(* CoDeSys 2.3 library: TcMC2.lib *)
(* Libraries: STANDARD.LIB 5.6.98 11:03:02, TcBase.lib*14.5.09 11:14:08, TcSystem.lib*15.1.10 08:10:33, TcBaseMath.lib 27.7.04 11:07:56, TcMath.lib 23.9.04 14:15:30 *)

(* Global variable list: TcMC_GlobalConstants *)
VAR_GLOBAL
	TcMcGlobal : _TCMCGLOBAL;
END_VAR
VAR_GLOBAL CONSTANT
	DEFAULT_HOME_POSITION 	:	LREAL 	:= 1.0E307;
END_VAR

(* Data type *)
{library private}
TYPE _E_ParameterType :
 (
	PARAMETERTYPE_NOTYPE := 0,
	PARAMETERTYPE_BOOL,
	PARAMETERTYPE_DWORD,
	PARAMETERTYPE_LREAL
 );
END_TYPE

(* Data type *)
{library private}
TYPE _E_ReadWriteParameterMode :
 (
	READWRITEPARAMETERMODE_READ 	:=10,
	READWRITEPARAMETERMODE_WRITE	:= 11
 );
END_TYPE

(* Data type *)
{library private}
TYPE _E_TcMC_STATES :
 (
	STATE_INITIALIZATION  := 100,
	STATE_ORDER,
	STATE_RUNNING,
	STATE_WAITING,
	STATE_MOTIONCOMMANDSLOCKED
 );
END_TYPE

(* Data type *)
TYPE _E_TcNC_CmdState :
 (
	CMDSTATE_SUCCESSFULLY_EXECUTED				:= 1,	(* bit number *)
	CMDSTATE_ABORTED_WITHOUT_ERROR				:= 2,
	CMDSTATE_ENDED_WITH_ERROR					:= 3,
	CMDSTATE_LASTCMD_SUCCESSFULLY_EXECUTED	:= 8,
	CMDSTATE_LASTCMD_ABORTED_WITHOUT_ERROR	:= 9,
	CMDSTATE_LASTCMD_ENDED_WITH_ERROR			:= 10
 );
END_TYPE

(* Data type *)
TYPE _E_TcNC_CmdTypeNewTargPosAndVelo :
 (
	TCNC_CHANGE_POS						:=  1,		(*Position (instantan)*)
	TCNC_CHANGE_VELO,							(*Geschwindigkeit (instantan)*)
	TCNC_CHANGE_POSANDVELO,					(*Position und Geschwindigkeit (instantan)*)
	TCNC_CHANGE_POS_AT_SWITCHPOS		:=  9,		(*Position (Umschaltposition)*)
	TCNC_CHANGE_VELO_AT_SWITCHPOS,			(*Geschwindigkeit (Umschaltposition)*)
	TCNC_CHANGE_POSANDVELO_AT_SWITCHPOS,	(*Position und Geschwindigkeit (Umschaltposition)*)
	TCNC_REACH_VELO_AT_POS				:= 14		(*neue Geschwindigkeit wird an einer bestimmten Position erreicht *)
 );
END_TYPE

(* Data type *)
TYPE _E_TcNC_PosSetType : (* mode is used with MC_SetPosition *)
(
	TCNC_POSSETTYPE_ABSOLUTE		:= 1,	(*Absolute position*)
	TCNC_POSSETTYPE_RELATIVE			(*Relative position*)
);
END_TYPE

(* Data type *)
TYPE _E_TcNC_ServoState :
 (
	TCNC_INACTIVE 	:= 0,
	TCNC_RUNNING,
	TCNC_OVERRIDE_ZERO,
	TCNC_PHASE_VELOCONST,
	TCNC_PHASE_ACCPOS,
	TCNC_PHASE_ACCNEG
 );
END_TYPE

(* Data type *)
TYPE _E_TcNC_SlaveTypes :
(
	TCNC_SLAVETYPE_LINEAR							:=	1,	(* Lineare Kopplung (Geradengleichung) *)
	TCNC_SLAVETYPE_FLYINGSAW_ONVELOCITY		:= 	2,	(* diagonal synchron. Aufkoppeln schnellstens auf Geschwindigkeit *)
	TCNC_SLAVETYPE_FLYINGSAW_ONPOSITION		:=	3,	(* diagonal synchron. Aufkoppeln auf Position und Geschwindigkeit *)
	TCNC_SLAVETYPE_FLYINGSAW_QUADRATIC		:=	4,	(* diagonal synchron. Aufkoppeln (quadratisches Geschw.-Profil) *)
	TCNC_SLAVETYPE_SYNCHRONIZING_ONVELO		:= 	5,	(* synchron. Aufkoppeln instantan auf Geschwindigkeit *)
	TCNC_SLAVETYPE_SYNCHRONIZING_ONPOS       	 	:= 	6,	(* synchron. Aufkoppeln auf Positionen und Geschwindigkeit *)
	TCNC_SLAVETYPE_SYNCJERKSETTER_ONVELO       	:= 	7,	(* synchron. Aufkoppeln auf Geschwindigkeit (zeitbasiert mittels Ruck-Steller) *)
	TCNC_SLAVETYPE_TABULAR						:=	10,	(* Tabellen-Kopplung ("simple/standard tabular slave") *)
	TCNC_SLAVETYPE_MULTITABULAR					:= 	11,	(* Tabellen-Kopplung ("multiscalable multi-tabular slave") *)
	TCNC_SLAVETYPE_FLYINGMODULO_LINEAR			:=	12,	(* Modulo Kopplung auf Position und/oder Geschwindigkeit mit anschliessender Linear Kopplung ("Schuette") *)
	TCNC_SLAVETYPE_MOTIONFUNCTIONTABULAR		:=	13,	(* Tabellen-Kopplung "motion functions" *)
	TCNC_SLAVETYPE_UNIVERSALTABULAR			:=	14,	(* Tabellen-Kopplung, universal tabular type substitues TABULAR, MULTITABULAR and MOTIONFUNCTION - 08.07.05 *)
	TCNC_SLAVETYPE_LINEAR_CYCLICCHANGES_RAMP	:=	15,	(* Lineare Kopplung (Geradengleichung) mit zyklischer Koppelfaktoraenderung *)
	TCNC_SLAVETYPE_BILINEAR						:=	16,	(* 27.04.01: Zweifach Lineare Kopplung (Geradengleichung)*)
	TCNC_SLAVETYPE_LINEAR_MULTIMASTER		:=	17,	(* 29.05.08: Lineare Multi-Master-Kopplung ('MC_GearInMultiMaster') *)
	TCNC_SLAVETYPE_CONST_SURFACEVELO_RAMP	:=	18	(* Verrechnete Winkelgeschwindigkeit fuer konstante Oberflaechengeschwindig. in Abhaengigkeit vom Radiusistwert des Enc.2 *)
);
END_TYPE

(* Data type *)
TYPE _E_TcNC_StartPosType :
(
	TCNC_START_ABSOLUTE					:= 1,		(*Start to absolute position*)
	TCNC_START_RELATIVE		,						(*Start to relative position*)
	TCNC_START_ENDLESS_PLUS	,					(*Start to endless positive position*)
	TCNC_START_ENDLESS_MINUS,						(*Start to endless negative position*)
	TCNC_START_MODULO,								(*Start to modulo position *)
	TCNC_START_ADDITIVE,								(*Start to a position relative to the last recent target position *)
	TCNC_START_MODULO_SHORT				:= 261, 	(*Start to modulo position *)
 	TCNC_START_MODULO_PLUS				:= 517, 	(*Start to modulo position *)
 	TCNC_START_MODULO_MINUS				:= 773, 	(*Start to modulo position *)
	TCNC_START_MODULO_CURRENT			:= 1029,	(* start to modulo position in current direction *)
 	TCNC_START_ABS_INTERNAL				:= 9, 		(*Start to absolute position, internal use*)
	TCNC_START_ENDLESSPLUS_SLOWMANUAL	:= 272,	(* manual jog mode *)
	TCNC_START_ENDLESSMINUS_SLOWMANUAL	:= 273,	(* manual jog mode *)
	TCNC_START_ENDLESSPLUS_FASTMANUAL	:= 528,	(* manual jog mode *)
	TCNC_START_ENDLESSMINUS_FASTMANUAL	:= 529,	(* manual jog mode *)
	TCNC_START_STOPANDLOCK				:= 4096,	(* stop axis and lock against any motion commands *)
	TCNC_START_HALT							:= 8192	(* halt axis - can be interrupted by any motion commands *)
);
END_TYPE

(* Data type *)
TYPE _E_TcNC_TargPosType :
(
	TCNC_POS_ABSOLUTE		:= 1,	(*Absolute position*)
	TCNC_POS_RELATIVE,			(*Relative position*)
	TCNC_POS_MODULO			:= 5,	(*Modulo position*)
	TCNC_POS_ABS_INTERNAL	:= 9	(*Absolute position, internal use*)
);
END_TYPE

(* Data type *)
(* MC_TouchProbe internal probe states *)
TYPE _E_TouchProbeState :
 (
	TouchProbeInactive,
	TouchProbeActivated,
	TouchProbeAborted
 );
END_TYPE

(* Data type *)
TYPE _ST_FunctionBlockResults :
STRUCT
	Done				:	BOOL;
	CommandAborted		:	BOOL;
	Error				:	BOOL;
	ErrorID				:	UDINT;
END_STRUCT
END_TYPE

(* Data type *)
TYPE _ST_NCADS_Axis :
STRUCT
	Parameter	:	_ST_NCADS_AxisParameter;
	State		:	_ST_NCADS_AxisState;
	Functions	:	_ST_NCADS_AxisFunctions;
END_STRUCT
END_TYPE

(* Data type *)
TYPE _ST_NCADS_AxisFunctions :
STRUCT
	IDXGRP		:	UDINT := 16#4200;
	IDXOFFS	:	_ST_NCADS_IDXOFFS_AxisFunctions;
END_STRUCT
END_TYPE

(* Data type *)
TYPE _ST_NCADS_AxisParameter :
STRUCT
	IDXGRP		:	UDINT := 16#4000;
	IDXOFFS	:	_ST_NCADS_IDXOFFS_AxisParameter;
END_STRUCT
END_TYPE

(* Data type *)
TYPE _ST_NCADS_AxisState :
STRUCT
	IDXGRP		:	UDINT := 16#4100;
	IDXOFFS	:	_ST_NCADS_IDXOFFS_AxisState;
END_STRUCT
END_TYPE

(* Data type *)
TYPE _ST_NCADS_IDXOFFS_AxisFunctions :
STRUCT
	RESET					: UDINT := 16#0001;
	STOP					: UDINT := 16#0002;
	CLEAR					: UDINT := 16#0003;
	EMERGENCYSTOP		: UDINT := 16#0004;
	PARAMETRIZEDSTOP	: UDINT := 16#0005;
	INITIALIZE				: UDINT := 16#0007;	(* Initialize Axis *)
	ORIENTEDSTOP			: UDINT := 16#0009;	(* 19.04.04 issue #2470 *)
	CALIBR					: UDINT := 16#0010;
	NEWTARGPOS			: UDINT := 16#0011;
	NEWTARGPOSANDVELO	: UDINT := 16#0012;
	CHANGEDYNAMICPARAM	: UDINT := 16#0015;	(* NEU: Neue Dynamikparameter (Acc;Dec) fuer Positionierung *)
	UNIVERSALSTART		: UDINT := 16#0016;	(* 05.03.07: new 'axis start and restart' command with buffer mode (issue #2786+#3276) *)
	SLAVEUNIVERSALSTART	: UDINT := 16#0017;	(* 24.02.09: decoupling command with succeding universal axis start commanded to a slave axis *)
(*	ONLINESTART			: UDINT := 16#0017;*)	(* 05.03.07: new 'axis start and restart' command (online start) (issue #2786+#3276) *)
	SETEXTERNALERROR	: UDINT := 16#0019;	(* 06.10.04: Externen Achsfehler setzen (Laufzeitfehler) issue #2665 *)
	SETPOS					: UDINT := 16#001A;
	SETCALFLAG			: UDINT := 16#001B;	(* "ist referenziert"-Flag setzen *)
	SETACTPOS				: UDINT := 16#001C;	(* nur Istwertsetzen ohne Sollwertaenderung !!! *)
	SETDRIVEPOS			: UDINT := 16#001D;	(* antriebsseitiges Istwertsetzen *)
	SETENCODERSCALING	: UDINT := 16#001E;	(* 17.07.08: "Fliegende Änderung des Skalierungsfaktors" *)
	SETPOSONTHEFLY		: UDINT := 16#001F;	(* 29.11.05: "Fliegendes Istwert Setzen" (betrifft Ist - und Sollwert) (issue #3017) *)
	START					: UDINT := 16#0020;
	STARTEXT				: UDINT := 16#0021;
	STARTVELOCHANGE		: UDINT := 16#0022;	(* special function for MMW *)
	ENABLEEXTGEN			: UDINT := 16#0023;	(* enable/start external setpoint values *)
	DISABLEEXTGEN			: UDINT := 16#0024;	(* disable/stop external setpoint values *)
	REVERSINGSEQUENCE	: UDINT := 16#0025;
	STARTDRVOUT			: UDINT := 16#0026;
	STOPDRVOUT			: UDINT := 16#0027;
	CHANGEDRVOUT		: UDINT := 16#0028;
	JUMPTOOVERRIDE		: UDINT := 16#0029;	(* 04.11.04: jump to actual override value and froze them until change (issue #2697) *)
(*	SETABSOLUTEMEASURING: UDINT := 16#002A;	removed 20091106 KSt *)	(* 29.11.05: "Fliegendes Istwert Setzen" (betrifft Ist - und Sollwert) (issue #3017) *)
	STARTSCOM			: UDINT := 16#0030;	(* 21.12.04: nun auch als 'ReadWrite'-Kommando *)
	STOPSCOM				: UDINT := 16#0031;
	CPL						: UDINT := 16#0040;	(* Achse koppeln *)
	DECPL					: UDINT := 16#0041;	(* Achse entkoppeln (und optional neue Endposition mit neuer Geschwindigkeit) *)
	CPLCHANGE				: UDINT := 16#0042;	(* Achse Koppelparams ändern *)
	TABCPLCHANGE			: UDINT := 16#0043;	(* 3x TabSlaveAxe Tabelle-Koppelparams ändern *)
	STOPSLAVE				: UDINT := 16#0044;	(* Slave-Stop (Diagonal-Slave / Flying Saw) *)
	CPLTAB					: UDINT := 16#0045;	(* TabSlaveAxe Koppelparams setzen *)
	TABSLVACTIVCOR		: UDINT := 16#0046;	(* 2x TabSlaveAxe Korrekturtabelle aktivieren (mit/ohne Aktivierungsposition) *)
	TABSLVLEAVECYC		: UDINT := 16#0047;	(* TabSlaveAxe	Monozyklische Tabelle beenden *)
	TABSLVCOROFFSET		: UDINT := 16#0048;	(* TabSlaveAxe	Letzter Korrektur Offset *)
	TABSLVSCALING			: UDINT := 16#0049;	(* NEU: Slave-Skalierung der Solo-Tabellenkopplung setzen *)
	CPLSOLOTAB			: UDINT := 16#004A;	(* Solo Tabellen Kopplung *)
	CPLSYNCHRONIZING		: UDINT := 16#004B;	(* Slave Synchronizing Generator ('GearInPos' and 'GearInVelo') *)
	CAMSCALING			: UDINT := 16#004D;	(* Slave Change CAM Scaling (Aenderung der Tabellenskalierung) (issue #2514) *)
	DISABLE				: UDINT := 16#0050;	(* Achse sperren *)
	ENABLE					: UDINT := 16#0051;	(* Achse reaktivieren *)
	CHANGEAXISCTRLLOOP	: UDINT := 16#0052;	(* NEU: Aenderung des aktiven Achsregelkreises *)
	DRIVEDISABLE			: UDINT := 16#0060;	(* Drive-Output der Achse sperren *)
	DRIVEENABLE			: UDINT := 16#0061;	(* Drive-Output der Achse reaktivieren *)
	RELEASEBRAKE			: UDINT := 16#0062;	(* Feststellbremse loesen (Eil/Schleich-Gruppe) *)
	RECONFIGURATE		: UDINT := 16#0070;	(* Achse zurueckfuehren in eigene PTP-Gruppe *)
END_STRUCT
END_TYPE

(* Data type *)
TYPE _ST_NCADS_IDXOFFS_AxisParameter :
STRUCT
	(* NC ADS Index Offsets for Axis Parameters *)
	PARAMSTRUCT				: UDINT := 16#0000;
	ID							: UDINT := 16#0001;
	NAME						: UDINT := 16#0002;
	AXISTYPE					: UDINT := 16#0003;
	CYCLETIME					: UDINT := 16#0004;
	UNITNAME					: UDINT := 16#0005;
	VELOREFSEARCH			: UDINT := 16#0006;
	VELOSYNCSEARCH			: UDINT := 16#0007;
	VELOSLOWMANUAL			: UDINT := 16#0008;
	VELOFASTMANUAL			: UDINT := 16#0009;
	VELOFAST					: UDINT := 16#000A;
	POSAREAENABLE			: UDINT := 16#000F;
	POSAREARANGE			: UDINT := 16#0010;
	MOTCNTRLENABLE			: UDINT := 16#0011;
	MOTCNTRLTIME				: UDINT := 16#0012;
	LOOPENABLE				: UDINT := 16#0013;
	LOOPDISTANCE				: UDINT := 16#0014;
	TARGETPOSENA			: UDINT := 16#0015;
	TARGETPOSRANGE			: UDINT := 16#0016;
	TARGETPOSTIME			: UDINT := 16#0017;
	PULSDISTPOS				: UDINT := 16#0018;
	PULSDISTNEG				: UDINT := 16#0019;
	UNITFLAGS					: UDINT := 16#0026;
	VELOMAXIMUM				: UDINT := 16#0027;
	MOTCNTRLRANGE			: UDINT := 16#0028;
	PEHCONTROLENA			: UDINT := 16#0029;
	PEHCONTROLTIME			: UDINT := 16#002A;
	BACKLASHCOMPENA			: UDINT := 16#002B;
	BACKLASH					: UDINT := 16#002C;
	DATAPERSISTENCE			: UDINT := 16#0030;
	HWAMSADDR				: UDINT := 16#0031;
	HWCHNNO					: UDINT := 16#0032;
	ACC							: UDINT := 16#0101;
	DEC						: UDINT := 16#0102;
	JERK						: UDINT := 16#0103;
	DELAY						: UDINT := 16#0104;
	OVERRIDETYPE				: UDINT := 16#0105;
	VELOJUMPFACTOR			: UDINT := 16#0106;
	REDUCTIONFEEDBACK		: UDINT := 16#0107;
	TOLERANCEBALLAUXAXIS	: UDINT := 16#0108;
	MAXPOSDEVIATIONAUXAXIS 	: UDINT := 16#0109;
	REF_POS					: UDINT := 16#0001_0103;
(*
	SCALE						= TCNC_IDXOFFS_AXmappedENC | 0x00000006;	// 0x00010006;
	ENABLESOFTENDMIN		= TCNC_IDXOFFS_AXmappedENC | 0x0000000B;	// 0x0001000B;
	ENABLESOFTENDMAX		= TCNC_IDXOFFS_AXmappedENC | 0x0000000C;	// 0x0001000C;
	SOFTENDMIN				= TCNC_IDXOFFS_AXmappedENC | 0x0000000D;	// 0x0001000D;
	SOFTENDMAX				= TCNC_IDXOFFS_AXmappedENC | 0x0000000E;	// 0x0001000E;
	ENABLEPOSDIFF				= TCNC_IDXOFFS_AXmappedCTR | 0x00000010;	// 0x00020010;
	POSDIFFMAX				= TCNC_IDXOFFS_AXmappedCTR | 0x00000012;	// 0x00020012;
	GAINPOS					= TCNC_IDXOFFS_AXmappedCTR | 0x00000102;	// 0x00020102;
	VELOREF					= TCNC_IDXOFFS_AXmappedDRV | 0x00000101;	// 0x00030101;
*)
END_STRUCT
END_TYPE

(* Data type *)
TYPE _ST_NCADS_IDXOFFS_AxisState :
STRUCT
	ONLINESTRUCT					: UDINT := 16#0000;
	ERROR							: UDINT := 16#0001;
(*
	ACTPOS							= TCNC_IDXOFFS_AXmappedENC | 0x00000002;	// 0x00010002;
	ACTVELO						= TCNC_IDXOFFS_AXmappedENC | 0x00000005;	// 0x00010005;
	ACTACC							= TCNC_IDXOFFS_AXmappedENC | 0x00000006;	// 0x00010006;
	MODULOACTPOS				= TCNC_IDXOFFS_AXmappedENC | 0x00000003;	// 0x00010003;
	MODULOACTTURNS				= TCNC_IDXOFFS_AXmappedENC | 0x00000004;	// 0x00010004;
	ACTINCREMENTS				= TCNC_IDXOFFS_AXmappedENC | 0x00000007;	// 0x00010007;
*)
	SETTASKCYCLE					: UDINT := 16#0009;
	SETPOS							: UDINT := 16#000A;
	SETVELO						: UDINT := 16#000E;
	SETACC							: UDINT := 16#000F;
	MODULOSETPOS				: UDINT := 16#000B;
	MODULOSETTURNS				: UDINT := 16#000C;
	SETDIR							: UDINT := 16#000D;
	TARGETPOSITION				: UDINT := 16#0013;
	REMAININGTIMEANDPOS			: UDINT := 16#0014;
	SETTASKCYCLE_WITHOUTCORR	: UDINT := 16#0019;
	SETPOS_WITHOUTCORR			: UDINT := 16#001A;
	SETVELO_WITHOUTCORR		: UDINT := 16#001E;
	SETACC_WITHOUTCORR			: UDINT := 16#001F;
	SETDIR_WITHOUTCORR			: UDINT := 16#001D;
	COUPLESTATE					: UDINT := 16#0020;
	CPLPARAMS						: UDINT := 16#0022;
	CPLFACTOR						: UDINT := 16#0023;
	AXISCTRLLOOPIDX				: UDINT := 16#0024;
	AXISSETPOINTGENIDX			: UDINT := 16#0025;
	CPLCHARACVALUES				: UDINT := 16#0026;
	CAMINFO						: UDINT := 16#0027;
(*
	POSDIFF						= TCNC_IDXOFFS_AXmappedCTR | 0x0000000F;	// 0x0002000F;
*)
END_STRUCT
END_TYPE

(* Data type *)
TYPE _ST_NCADS_IDXOFFS_TableFunctions :
STRUCT
	(* Index Offset definitions of table functions *)
	CREATETAB				: UDINT := 	16#0001_0000;		(* create table*)
	CREATEMOTIONTAB 		: UDINT := 	16#0001_0010;		(* create motion function table*)
	DELETETAB 				: UDINT := 	16#0002_0000; 		(* delete tables *)
END_STRUCT
END_TYPE

(* Data type *)
TYPE _ST_NCADS_IDXOFFS_TableParameter :
STRUCT
	MFREADCHARACVALUES	: UDINT := 	16#0000_0050;		(* read characteristic values of a motion function *)
	WRITETABROWS 		: UDINT := 	16#0100_0000;		(* write table *)
(*	WRITETABCOLS 			: UDINT := 	16#0200_0000;	*)	(* write table *)
	WRITEMFTABROWS 		: UDINT := 	16#0500_0000;		(* write motion function table *)
(*	WRITEMFTABCOLS 		: UDINT := 	16#0600_0000;	*)	(* write motion function table *)
(*	READSLAVEPOS 		: UDINT := 	16#0000_0021;	*)	(* read slave table position related to a master position *)
	MFREADTAB 			: UDINT := 	16#0000_0022;		(* read motion function as data table *)
	READSLAVEDYNAMICS 	: UDINT := 	16#0000_0023;		(* read slave table position, velocity and acceleration related to a master position *)
	READMASTERPOSITION 	: UDINT := 	16#0000_0024;		(* read master table position related  to slave position *)
END_STRUCT
END_TYPE

(* Data type *)
TYPE _ST_NCADS_Table :
STRUCT
	Parameter	:	_ST_NCADS_TableParameter;
	Functions	:	_ST_NCADS_TableFunctions;
END_STRUCT
END_TYPE

(* Data type *)
TYPE _ST_NCADS_TableFunctions :
STRUCT
	IDXGRP		:	UDINT := 16#A200;
	IDXOFFS	:	_ST_NCADS_IDXOFFS_TableFunctions;
END_STRUCT
END_TYPE

(* Data type *)
TYPE _ST_NCADS_TableParameter :
STRUCT
	IDXGRP		:	UDINT := 16#A000;
	IDXOFFS	:	_ST_NCADS_IDXOFFS_TableParameter;
END_STRUCT
END_TYPE

(* Data type *)
{library private}
TYPE _ST_ParaStruct :
STRUCT
	IndexGroup 	:	UDINT;
	IndexOffset 	:	UDINT;
	ParaType	:	_E_ParameterType;
	LrealSize	:	UDINT; (* sizeof Lreal data array *)
	LrealOffset	: 	UDINT; (* offset in lreal data array *)
END_STRUCT
END_TYPE

(* Data type *)
TYPE _ST_TcNC_Compensation2 :	(* internal use with MC_MoveSuperimposed_2 *)
STRUCT
	nCompType	:	UDINT;	(* E_SuperpositionMode *)
	fAccPlus		:	LREAL;
	fAccMinus	:	LREAL;
	fVeloDiff		:	LREAL;
	fVeloProcess	:	LREAL;
	fDistance	:	LREAL;	(* distance to compensate *)
	fLength		:	LREAL;	(* distance moved during compensation *)
	nWarningId	: 	UDINT;	(* documented as error code *)
END_STRUCT
END_TYPE

(* Data type *)
TYPE _ST_TcNC_CoupleSlave :
STRUCT
	nSlaveType		:	UDINT;
	nMasterAxisId	:	UDINT;
	nMasterSubIdx	:	UDINT;
	nSlaveSubIdx	:	UDINT;
	fCoupleParam1	:	LREAL;
	fCoupleParam2	:	LREAL;
	fCoupleParam3	:	LREAL;
	fCoupleParam4	:	LREAL;
END_STRUCT
END_TYPE

(* Data type *)
TYPE _ST_TcNC_CoupleSlaveMultiMaster :
STRUCT
	nSlaveType		:	UDINT;
	nMasterAxisId	:	UDINT;
	nMasterSubIdx	:	UDINT;
	nSlaveSubIdx		:	UDINT;
(*	nMasterID1 = nMasterAxisId *)
	nMasterID2		:	UDINT;
	nMasterID3		:	UDINT;
	nMasterID4		:	UDINT;
	nMasterID5		:	UDINT;
	nMasterID6		:	UDINT;
	nMasterID7		:	UDINT;
	nMasterID8		:	UDINT;
	fSlaveAcceleration:	LREAL;
	nCheckAndOpMode:	DWORD;
END_STRUCT
END_TYPE

(* Data type *)
TYPE _ST_TcNC_DecoupleSlave :
STRUCT
	nDecoupleMode	:	UDINT;
	fNewPosEnd	:	LREAL;
	fNewVeloRequ	:	LREAL;
	fAcceleration	:	LREAL;
	fDeceleration	:	LREAL;
	fJerk			:	LREAL;
END_STRUCT
END_TYPE

(* Data type *)
TYPE _ST_TcNc_OperationModes :
STRUCT
	(* OpModeDWord in cyclic interface *)
	PosAreaControl	:	DWORD := 2#0000_0000_0000_0000_0000_0000_0000_0001;
	TargetPosControl	:	DWORD := 2#0000_0000_0000_0000_0000_0000_0000_0010;
	AllowSlaveCommands :DWORD	:= 2#0000_0000_0010_0000_0000_0000_0000_0000;
	(*
	Loop			:	DWORD := 2#0000_0000_0000_0000_0000_0000_0000_0100;
	MotionControl		:	DWORD := 2#0000_0000_0000_0000_0000_0000_0000_1000;
	PEHTimeControl	:	DWORD := 2#0000_0000_0000_0000_0000_0000_0001_0000;
	BacklashComp	:	DWORD := 2#0000_0000_0000_0000_0000_0000_0010_0000;
	*)
	(* bits 6 .. 15 reserved *)
	(*
	PosDiffControl  	:	DWORD := 2#0000_0000_0000_0001_0000_0000_0000_0000;
	VeloDiffControl	:	DWORD := 2#0000_0000_0000_0010_0000_0000_0000_0000;
	SoftEndMinControl	:	DWORD := 2#0000_0000_0000_0100_0000_0000_0000_0000;
	SoftEndMaxControl	:	DWORD := 2#0000_0000_0000_1000_0000_0000_0000_0000;
	ActPosCorrection	:	DWORD := 2#0000_0000_0001_0000_0000_0000_0000_0000;
	*)
	(* bits 21 .. 31 reserved *)
END_STRUCT
END_TYPE

(* Data type *)
TYPE _ST_TcNC_SetEncoderSaclingFactor :
STRUCT
 	nEncoderScalingFactorType	:	UINT;
	nCtrlWord					:	UINT; 	(* additional option flags *)	(* added KSt 2009-04-09 *)
	fEncoderScalingFactor			:	LREAL;
END_STRUCT
END_TYPE

(* Data type *)
TYPE _ST_TcNC_SetPos :
STRUCT
	nPosIstType		:	UDINT;
	fNewPosIst		:	LREAL;
END_STRUCT
END_TYPE

(* Data type *)
TYPE _ST_TcNC_SetPosOnTheFly :
STRUCT
	nPosSetType		: 	UDINT; 	(*_E_TcNC_PosSetType *)	(* Absolute, Relative - added KSt 2009-01-28 *)
	nCtrlDWord		:	UDINT; 	(* additional option flags *)	(* added KSt 2009-01-28 *)
 	fPreviousActualPos:	LREAL;	(* value not used any longer since 2009-01-28 *)
	fNewActualPos	:	LREAL;
	nReserved		:	ARRAY[1..2] OF DWORD;	(* added KSt 2009-01-28 *)
END_STRUCT
END_TYPE

(* Data type *)
TYPE _ST_TcNC_UnversalAxisStartRequest :
STRUCT
	nStartType	: UDINT;			(* axis start TYPE (ABSOLUT, RELATIV, ENDLESS_PLUS, ENDLESS_MINUS, MODULO_SHORT, MODULO_PLUS, MODULO_MINUS) *)
	nControlMask	: UDINT;			(* optional: control mask *)

	fPosTarget	: LREAL;			(* target position *)
	fVeloRequ	: LREAL;			(* required velocity *)

	fAcc			: LREAL;			(* acceleration (>= 0) *)
	fDec		: LREAL;			(* deceleration (>= 0) *)
	fJerk		: LREAL;			(* jerk (>= 0) *)

	nBufferMode	: UDINT;			(* optional: 'buffer mode' OR 'activation mode' FOR 'buffered commands' (issue #2786) *)
	fBlendingPosition: LREAL;			(* optional: activation position *)

	fVeloStart	: LREAL;			(* optional: start velocity	(0 <= fVeloStart <= fVeloRequ)	Frage: erstmal weglassen ??? *)
	fVeloEnd		: LREAL;			(* optional: end velocity		(0 <= fVeloEnd <= fVeloRequ)	Frage: erstmal weglassen ??? *)
END_STRUCT
END_TYPE

(* Data type *)
TYPE _ST_TcNC_UnversalAxisStartResponse :
STRUCT
	nCmdNo 	: WORD;			(* Continuous actual command number *)
	nCmdState	: WORD;			(* Command state *)
END_STRUCT
END_TYPE

(* Data type *)
TYPE AXIS_REF : _FBAXIS_REF;
END_TYPE

(* Data type *)
(* for details: see TwinCAT Information System*)
TYPE E_AxisErrorCodes : (
		MC_ERROR_NO_ERROR := 0,
(*		MC_ERROR_NO_ORDER,		deleted 15.07.2005 KSt *)
(*		MC_ERROR_OVERRIDE,		deleted 15.07.2005 KSt *)
(*		MC_ERROR_LOW_VELOCITY,	deleted 15.07.2005 KSt *)
		MC_ERROR_AXIS_HAS_BEEN_STOPPED		:= 16#4B00,
		MC_ERROR_AXIS_CAN_NOT_BE_STARTED	:= 16#4B01,
		MC_ERROR_CONTROLMODE_NOT_ALLOWED	:= 16#4B02,
		MC_ERROR_AXIS_IS_NOT_MOVING			:= 16#4B03,
		MC_ERROR_WRONG_MODE					:= 16#4B04,
		MC_ERROR_COMMAND_NOT_ALLOWED		:= 16#4B05,
		MC_ERROR_PARAMETER_NOT_CORRECT		:= 16#4B06,
		MC_ERROR_TARGETPOS_TIMEOUT			:= 16#4B07,
		MC_ERROR_AXIS_IN_PROTECTED_MODE		:= 16#4B08,
		MC_ERROR_AXIS_IS_NOT_READY				:= 16#4B09,
		MC_ERROR_CALIBRATION_ERROR			:= 16#4B0A,
		MC_ERROR_INVALID_TOUCH_PROBE			:= 16#4B0B,
		MC_ERROR_TOUCH_PROBE_DEACTIVATED	:= 16#4B0C,
		MC_ERROR_SUPPLEMENT_NOT_INSTALLED	:= 16#4B0E,
		(*======================================================================	*)
		(*	4B0F 	timeout terminal register access									*)
		(*======================================================================	*)
		(* 	4B10 .. 4B2F used in NCI context 											*)
		(*======================================================================	*)
		(* 	4B30 .. 4B3F used in TcMcCam - MC_NC_TableErrorCodes					*)
		(*======================================================================	*)
		(* 	4B40 .. 4B4F used in TcNc for programming KL25xx terminals 					*)
		(*======================================================================	*)
		(* 	4B50 .. 4B5F used in TcRemoteSync.lib									*)
		(*======================================================================	*)
		(* 	4B60 .. 4B6F used in TcMC for buffered commands  *)
		MC_ERROR_BUFFERED_COMMAND_NOT_STARTED			:= 16#4B60,
		MC_ERROR_BUFFERED_COMMAND_MONITORING_IMPOSSIBLE	:= 16#4B61,
		MC_ERROR_BUFFERED_COMMAND_ERRORID_NOT_AVAILABLE	:= 16#4B62,
		MC_ERROR_BUFFERED_COMMAND_NO_STATE_FEEDBACK		:= 16#4B63,
		MC_ERROR_BUFFERMODE_NOT_SUPPORTED					:= 16#4B64,
		MC_ERROR_BUFFERED_COMMAND_CMDNOZERO				:= 16#4B65,
		(*======================================================================	*)
		(* 	4B70 .. 4B7F used in TcMC for I/O related errors *)
		MC_ERROR_TERMINALFEEDBACK								:= 16#4B70
		(*======================================================================	*)
(*		MC_ERROR_FUNCTION_IS_BUSY := 16#4B99	*)
		);
END_TYPE

(* Data type *)
TYPE E_DestallDetectMode :
	(
		PwStDetectMode_None := 0,		(* do not detect stall situations *)
		PwStDetectMode_Encoderless,		(* use status signals of KL2531/KL2541 for stall detection *)
		PwStDetectMode_Lagging			(* use encoder signals for stall detection *)
	);
END_TYPE

(* Data type *)
TYPE E_DestallMode :
	(
		PwStMode_None := 0,			(* do not respond to stall situations *)
		PwStMode_SetError,			(* in stall situations place axis in fault state *)
		PwStMode_SetErrNonRef,		(* in stall situations place axis in nonreferenced state *)
		PwStMode_UseOverride			(* use override to catch the axis and recover from stall situations *)
	);
END_TYPE

(* Data type *)
TYPE E_JogMode :
 (
	MC_JOGMODE_STANDARD_SLOW,	(* motion with standard jog parameters for slow motion *)
	MC_JOGMODE_STANDARD_FAST,		(* motion with standard jog parameters for fast motion *)
	MC_JOGMODE_CONTINOUS,		 	(* axis moves as long as the jog button is pressed using parameterized dynamics *)
	MC_JOGMODE_INCHING,				(* axis moves for a certain relative distance *)
	MC_JOGMODE_INCHING_MODULO		(* axis moves for a certain relative distance - stop position is rounded to the distance value *)
 );
END_TYPE

(* Data type *)
TYPE E_PositionType :
(
	POSITIONTYPE_ABSOLUTE	:= 1,	(*Absolute position*)
	POSITIONTYPE_RELATIVE,		(*Relative position*)
	POSITIONTYPE_MODULO		:= 5	(*Modulo position*)
);
END_TYPE

(* Data type *)
TYPE E_ReadMode :
 (
 	READMODE_ONCE	:= 1,
	READMODE_CYCLIC
 );
END_TYPE

(* Data type *)
TYPE E_SetScalingFactorMode :
 (
	ENCODERSCALINGMODE_ABSOLUTE	:= 1,
	ENCODERSCALINGMODE_RELATIVE	:=2
 );
END_TYPE

(* Data type *)
(* signal edge used with MC_TouchProbe *)
TYPE E_SignalEdge :
 (
	RisingEdge,
	FallingEdge
 );
END_TYPE

(* Data type *)
TYPE E_SuperpositionAbortOption :
 (
 	SUPERPOSITIONOPTION_ABORTATSTANDSTILL := 0,	(* aborts the superposition when the subordinated motion profile velocity is zero - standard of  MC_MoveSuperimposed (TcMC version 1) *)
 	SUPERPOSITIONOPTION_RESUMEAFTERSTANDSTILL,	(* resumes the superposition after a temporary standstill of the subordinated motion profile *)
 	SUPERPOSITIONOPTION_RESUMEAFTERMOTIONSTOP	(* resumes the superposition after any stop and restart of the subordinated motion profile - ResumeAfterMotionStop includes ResumeAfterStandstill *)
 );
END_TYPE

(* Data type *)
TYPE E_SuperpositionMode :
 (
 	SUPERPOSITIONMODE_VELOREDUCTION_ADDITIVEMOTION := 1,	(* standard type of  MC_MoveSuperimposed (TcMC version 1) *)
 	SUPERPOSITIONMODE_VELOREDUCTION_LIMITEDMOTION,
 	SUPERPOSITIONMODE_LENGTHREDUCTION_ADDITIVEMOTION,
 	SUPERPOSITIONMODE_LENGTHREDUCTION_LIMITEDMOTION,
 	SUPERPOSITIONMODE_ACCREDUCTION_ADDITIVEMOTION,			(* new 2009-05 *)
 	SUPERPOSITIONMODE_ACCREDUCTION_LIMITEDMOTION			(* new 2009-05 *)
 );
END_TYPE

(* Data type *)
(* MC_TouchProbe probes *)
TYPE E_TouchProbe :
 (
	TouchProbe1 := 1,	(* hardware probe with AX2000, SERCOS, KL5xxx and others *)
	TouchProbe2,	(* currently not available *)
	TouchProbe3,	(* currently not available *)
	TouchProbe4,	(* currently not available *)
	PlcEvent := 10		(* simple PLC signal TRUE/FALSE *)
 );
END_TYPE

(* Data type *)
TYPE MC_AxisParameter : (
(*				PLCopen specific parameters *)			(* Index-Group 0x4000 + ID*)
				CommandedPosition := 1,		(* lreal *)	(* taken from NcToPlc *)
				SWLimitPos,					(* lreal *)	(* IndexOffset= 16#0001_000E *)
				SWLimitNeg,					(* lreal *)	(* IndexOffset= 16#0001_000D *)
				EnableLimitPos,				(* bool *)	(* IndexOffset= 16#0001_000C *)
				EnableLimitNeg,				(* bool *)	(* IndexOffset= 16#0001_000B *)
				EnablePosLagMonitoring,		(* bool *)	(* IndexOffset= 16#0002_0010 *)
				MaxPositionLag,				(* lreal *)	(* IndexOffset= 16#0002_0012 *)
				MaxVelocitySystem,			(* lreal *)	(* IndexOffset= 16#0000_0027 *)
				MaxVelocityAppl,				(* lreal *)	(* IndexOffset= 16#0000_0027 *)
				ActualVelocity,				(* lreal *)	(* taken from NcToPlc *)
				CommandedVelocity,			(* lreal *)	(* taken from NcToPlc *)
				MaxAccelerationSystem,		(* lreal *)	(* IndexOffset= 16#0000_0101 *)
				MaxAccelerationAppl,			(* lreal *)	(* IndexOffset= 16#0000_0101 *)
				MaxDecelerationSystem,		(* lreal *)	(* IndexOffset= 16#0000_0102 *)
				MaxDecelerationAppl,			(* lreal *)	(* IndexOffset= 16#0000_0102 *)
				MaxJerk,						(* lreal *)	(* IndexOffset= 16#0000_0103 *)

(*				Beckhoff specific parameters *)		 	(* Index-Group 0x4000 + ID*)
				AxisId	:=	1000,			(* lreal *)	(* IndexOffset= 16#0000_0001 *)
				AxisVeloManSlow,				(* lreal *)	(* IndexOffset= 16#0000_0008 *)
				AxisVeloManFast,				(* lreal *)	(* IndexOffset= 16#0000_0009 *)
				AxisVeloMax,					(* lreal *)	(* IndexOffset= 16#0000_0027 *)
				AxisAcc,						(* lreal *)	(* IndexOffset= 16#0000_0101 *)
				AxisDec,						(* lreal *)	(* IndexOffset= 16#0000_0102 *)
				AxisJerk,						(* lreal *)	(* IndexOffset= 16#0000_0103 *)
				AxisMaxVelocity,				(* lreal *)	(* IndexOffset= 16#0000_0027 *)
				AxisRapidTraverseVelocity,	(* lreal *)	(* IndexOffset= 16#0000_000A *)
				AxisManualVelocityFast,		(* lreal *)	(* IndexOffset= 16#0000_0009 *)
				AxisManualVelocitySlow,		(* lreal *)	(* IndexOffset= 16#0000_0008 *)
				AxisCalibrationVelocityForward,	(* lreal *)	(* IndexOffset= 16#0000_0006 *)
				AxisCalibrationVelocityBackward,(* lreal *)	(* IndexOffset= 16#0000_0007 *)
				AxisJogIncrementForward,		(* lreal *)	(* IndexOffset= 16#0000_0018 *)
				AxisJogIncrementBackward,	(* lreal *)	(* IndexOffset= 16#0000_0019 *)
				AxisEnMinSoftPosLimit,			(* bool *)	(* IndexOffset= 16#0001_000B *)
				AxisMinSoftPosLimit,			(* lreal *)	(* IndexOffset= 16#0001_000D *)
				AxisEnMaxSoftPosLimit,		(* bool *)	(* IndexOffset= 16#0001_000C *)
				AxisMaxSoftPosLimit,			(* lreal *)	(* IndexOffset= 16#0001_000E *)
				AxisEnPositionLagMonitoring,	(* bool *)	(* IndexOffset= 16#0002_0010 *)
				AxisMaxPosLagValue,			(* lreal *)	(* IndexOffset= 16#0002_0012 *)
				AxisMaxPosLagFilterTime,		(* lreal *)	(* IndexOffset= 16#0002_0013 *)
				AxisEnPositionRangeMonitoring,	(* bool *)	(* IndexOffset= 16#0000_000F *)
				AxisPositionRangeWindow,		(* lreal *)	(* IndexOffset= 16#0000_0010 *)
				AxisEnTargetPositionMonitoring,	(* bool *)	(* IndexOffset= 16#0000_0015 *)
				AxisTargetPositionWindow,		(* lreal *)	(* IndexOffset= 16#0000_0016 *)
				AxisTargetPositionMonitoringTime,(* lreal *)(* IndexOffset= 16#0000_0017 *)
				AxisEnInTargetTimeout,		(* bool *)	(* IndexOffset= 16#0000_0029 *)
				AxisInTargetTimeout,			(* lreal *)	(* IndexOffset= 16#0000_002A *)
				AxisEnMotionMonitoring,		(* bool *)	(* IndexOffset= 16#0000_0011 *)
				AxisMotionMonitoringWindow,	(* lreal *)	(* IndexOffset= 16#0000_0028 *)
				AxisMotionMonitoringTime,		(* lreal *)	(* IndexOffset= 16#0000_0012 *)
				AxisDelayTimeVeloPosition,	(* lreal *)	(* IndexOffset= 16#0000_0104 *)
				AxisEnLoopingDistance,		(* bool *)	(* IndexOffset= 16#0000_0013 *)
				AxisLoopingDistance,			(* lreal *)	(* IndexOffset= 16#0000_0014 *)
				AxisEnBacklashCompensation,	(* bool *)	(* IndexOffset= 16#0000_002B *)
				AxisBacklash,				(* lreal *)	(* IndexOffset= 16#0000_002C *)
				AxisEnDataPersistence,		(* bool *)	(* IndexOffset= 16#0000_0030 *)
				AxisRefVeloOnRefOutput,		(* lreal *)	(* IndexOffset= 16#0003_0101 *)
				AxisOverrideType,			(* lreal *)	(* IndexOffset= 16#0000_0105 *)
				(* new since 4/2007 *)
				AxisEncoderScalingFactor,		(* lreal *)	(* IndexOffset= 16#0001_0006 *)
				AxisEncoderOffset,			(* lreal *)	(* IndexOffset= 16#0001_0007 *)
				AxisEncoderDirectionInverse,	(* bool *)	(* IndexOffset= 16#0001_0008 *)
				AxisEncoderMask,			(* dword *)(* IndexOffset= 16#0001_0015 *)
				AxisEncoderModuloValue,		(* lreal *)	(* IndexOffset= 16#0001_0009 *)
				AxisModuloToleranceWindow,	(* lreal *)	(* IndexOffset= 16#0001_001B *)
				AxisEnablePosCorrection,		(* bool *)	(* IndexOffset= 16#0001_0016 *)
				AxisPosCorrectionFilterTime,	(* lreal *)	(* IndexOffset= 16#0001_0017 *)
				AxisUnitInterpretation,			(* lreal *)	(* IndexOffset= 16#0000_0026 *)	(* added 5/20/2008 KSt *)
				(* new since 1/2010 *)
				AxisMotorDirectionInverse,		(* bool *)	(* IndexOffset= 16#0003_0006 *)

(*				Beckhoff specific axis status information - READ ONLY *)	(* Index-Group 0x4100 + ID*)
				AxisTargetPosition	:= 2000,	(* lreal *)	(* IndexOffset= 16#0000_0013 *)
				AxisRemainingTimeToGo,		(* lreal *)	(* IndexOffset= 16#0000_0014 *)
				AxisRemainingDistanceToGo,	(* lreal *)	(* IndexOffset= 16#0000_0022, 16#0000_0042 *)

(*				Beckhoff specific axis functions *)
				AxisGearRatio		:= 3000	(* lreal *) 	(* read:IdxGrp=0x4100+ID, IdxOffs=16#0000_0022, read:IdxGrp=0x4200+ID, IdxOffs=16#0000_0042 *)	(* read/write gear ratio of a slave - added 6/08/2008 KSt *)
				);
END_TYPE

(* Data type *)
(* 	PLCopen axis states
	The axis states are defined in the PLCopen state diagram
*)
TYPE MC_AxisStates :
 (
	MC_AXISSTATE_UNDEFINED,
	MC_AXISSTATE_DISABLED,
	MC_AXISSTATE_STANDSTILL,
	MC_AXISSTATE_ERRORSTOP,
	MC_AXISSTATE_STOPPING,
	MC_AXISSTATE_HOMING,
	MC_AXISSTATE_DISCRETEMOTION,
	MC_AXISSTATE_CONTINOUSMOTION,
	MC_AXISSTATE_SYNCHRONIZEDMOTION
 );
END_TYPE

(* Data type *)
TYPE MC_BufferMode :
 (
	MC_Aborting			:= 16#00,
	MC_Buffered			:= 16#01,
	MC_BlendingLow		:= 16#12,
	MC_BlendingPrevious	:= 16#13,
	MC_BlendingNext		:= 16#14,
	MC_BlendingHigh		:= 16#15
 );
END_TYPE

(*	PLCopen Description

Aborting versus Buffered modes
Some of the FBs have an input called 'BufferMode'. With this input, the FB can either work in a ‘Non-buffered mode’
(default behavior) or in a ‘Buffered mode’. The difference between those modes is when they should start their action:
  -	A command in a non-buffered mode acts immediately, even if this interrupts another motion
  - 	A command in a buffered mode waits till the current FB sets its Done output (or InPosition, or InVelocity,..).

There are several options for the buffered mode. For this reason, this input is an ENUM of type MC_BUFFERMODE.
The following modes have been identified:

  -	Aborting 			Default mode without buffering. The next FB aborts an ongoing motion and the command
					affects the axis immediately.
  -	Buffered 			The next FB affects the axis as soon as the previous movement is Done There is no
					blending.
  -	BlendingLow 		The next FB controls the axis after the previous FB has finished (equivalent to buffered),
					but the axis will not stop between the movements. The velocity is blended with the lowest
					velocity of both commands (1 and 2) at the first end-position (1).
  -	BlendingPrevious 	blending with the velocity of FB 1 at end-position of FB 1
  -	BlendingNext 		blending with velocity of FB 2 at end-position of FB1
  -	BlendingHigh 	blending with highest velocity of FB 1 and FB 2 at end-position of FB1

*)

(* Data type *)
TYPE MC_Direction :
(
	MC_Positive_Direction := 1,
	MC_Shortest_Way ,
	MC_Negative_Direction,
	MC_Current_Direction
);
END_TYPE

(* Data type *)
TYPE MC_HomingMode :
 (
	MC_DefaultHoming,	(* default homing as defined in the SystemManager encoder parameters *)
	MC_AbsSwitch,		(* not implemented - Absolute Switch homing plus Limit switches *)
	MC_LimitSwitch,		(* not implemented - Homing against Limit switches *)
	MC_RefPulse,		(* not implemented - Homing using encoder Reference Pulse "Zero Mark" *)
	MC_Direct,			(* Static Homing forcing position from user reference *)
	MC_Absolute,			(* not implemented - Static Homing forcing position from absolute encoder *)
	MC_Block,			(* not implemented - Homing against hardware parts blocking movement *)
	MC_ForceCalibration,	(* set the calibration flag without performing any motion or changing the position *)
	MC_ResetCalibration	(* resets the calibration flag without performing any motion or changing the position *)
 );
END_TYPE

(* Data type *)
TYPE NCTOPLC_AXIS_REF
STRUCT
	StateDWord      			: DWORD;      	(* Status double word *)
    	ErrorCode          			: DWORD;      	(* Axis error code *)
    	AxisState     	    			: DWORD;      	(* Axis moving status *)
    	AxisModeConfirmation		: DWORD;      	(* Axis mode confirmation (feedback from NC) *)
    	HomingState   			: DWORD;      	(* State of axis calibration (homing) *)
    	CoupleState        			: DWORD;      	(* Axis coupling state *)
    	SvbEntries         			: DWORD;      	(* SVB entries/orders (SVB = Set preparation task) *)
    	SafEntries        			: DWORD;      	(* SAF entries/orders (SAF = Set execution task) *)
    	AxisId        				: DWORD;	(* Axis ID *)
    	OpModeDWord        		: DWORD;      	(* Current operation mode *)
	ActiveControlLoopIndex 	: WORD;	 	(* Active control loop index *)
	ControlLoopIndex 			: WORD;	 	(* Axis control loop index (0, 1, 2, when multiple control loops are used) *)
    	ActPos            				: LREAL;      	(* Actual position (absolut value from NC) *)
    	ModuloActPos      			: LREAL;      	(* Actual modulo position *)
    	ModuloActTurns  			: DINT;       	(* Actual modulo turns *)
    	ActVelo           				: LREAL;      	(* Actual velocity *)
    	PosDiff            				: LREAL;      	(* Position difference (lag distance) *)
    	SetPos	            			: LREAL;      	(* Setpoint position *)
    	SetVelo           				: LREAL;      	(* Setpoint velocity *)
	SetAcc					: LREAL; 		(* Setpoint acceleration *)
    	TargetPos    				: LREAL;      	(* Estimated target position *)
    	ModuloSetPos    			: LREAL;      	(* Setpoint modulo position *)
    	ModuloSetTurns    			: DINT;      	(* Setpoint modulo turns *)
    	CmdNo    				: WORD;		(* Continuous actual command number *)
    	CmdState    				: WORD;		(* Command state *)
END_STRUCT
END_TYPE

(* Data type *)
TYPE PLCTONC_AXIS_REF
STRUCT
	ControlDWord	: 	DWORD;	(* Control double word *)
	Override			: 	DWORD;	(* Velocity override *)
	AxisModeRequest : 	DWORD;	(* Axis operating mode (PLC request) *)
	AxisModeDWord	:	DWORD;	(* optional mode parameter *)
	AxisModeLReal	:	LREAL;		(* optional mode parameter *)
	PositionCorrection :	LREAL;		(* Correction value for current position *)
	ExtSetPos		:	LREAL;		(* external position setpoint *)
	ExtSetVelo		:	LREAL;		(* external velocity setpoint *)
	ExtSetAcc		:	LREAL;		(* external acceleration setpoint *)
	ExtSetDirection	: 	DINT;      		(*  external direction setpoint *)
	{library private}
	Reserved1		: 	DWORD;	(* reserved *)
	{library public}
	ExtControllerOutput :	LREAL;		(* external controller output *)
	GearRatio1		: 	LREAL;		(* Gear ratio for dynamic multi master coupling modes *)
	GearRatio2		: 	LREAL;		(* Gear ratio for dynamic multi master coupling modes *)
	GearRatio3		: 	LREAL;		(* Gear ratio for dynamic multi master coupling modes *)
	GearRatio4		: 	LREAL;		(* Gear ratio for dynamic multi master coupling modes *)
	{library private}
	MapState		:	BYTE;		(* reserved - internal use *)
	{library public}
	PlcCycleControl	:	BYTE;
	PlcCycleCount	:	BYTE;
	{library private}
	Reserved_HIDDEN    :	ARRAY [107..127] OF BYTE;
END_STRUCT
END_TYPE

(* Data type *)
TYPE ST_AdsAddress :
STRUCT
	NetId 	: STRING(23);
	Port 		: UINT;
	Channel 	: UINT;
END_STRUCT
END_TYPE

(* Data type *)
TYPE ST_AxisComponents :
STRUCT
	EncoderIDs	: ARRAY[1..9] OF DWORD;
	ControllerIDs 	: ARRAY[1..9] OF DWORD;
	DriveIDs 		: ARRAY[1..9] OF DWORD;
END_STRUCT
END_TYPE

(* Data type *)
(* axis operation mode feedback from NcToPlc. *)
TYPE ST_AxisOpModes :
STRUCT
	PositionAreaMonitoring 	: BOOL;	(* bit 0 - OpModeDWord *)
	TargetPositionMonitoring 	: BOOL;	(* bit 1 - OpModeDWord *)
	LoopMode				: BOOL;	(* bit 2 - OpModeDWord - loop mode for two speed axes *)
	MotionMonitoring			: BOOL;	(* bit 3 - OpModeDWord *)
	PEHTimeMonitoring		: BOOL;	(* bit 4 - OpModeDWord *)
	BacklashCompensation	: BOOL;	(* bit 5 - OpModeDWord *)
	DelayedErrorReaction		: BOOL;	(* bit 6 - OpModeDWord *)
	Modulo					: BOOL;	(* bit 7 - OpModeDWord - axis is parameterized as modulo axis *)
	PositionLagMonitoring		: BOOL;	(* bit 16 - OpModeDWord *)
	VelocityLagMonitoring		: BOOL;	(* bit 17 - OpModeDWord *)
	SoftLimitMinMonitoring		: BOOL;	(* bit 18 - OpModeDWord *)
	SoftLimitMaxMonitoring		: BOOL;	(* bit 19 - OpModeDWord *)
	PositionCorrection			: BOOL;	(* bit 20 - OpModeDWord *)
	AllowSlaveCommands		: BOOL;	(* bit 21 - OpModeDWord - allow motion commands on slave axes with automatic decoupling *) 	(* 2008-02-20 KSt *)
END_STRUCT
END_TYPE

(* Data type *)
TYPE ST_AxisParameterSet :
STRUCT
	(* AXIS: *)
	AxisId 						: DWORD;	(* 0x00000001 *)
	sAxisName 					: STRING(31);	(* 0x00000002 *)
	nAxisType					: DWORD;	(* 0x00000003 *)
	bEnablePositionAreaControl 	: WORD;		(* 0x0000000F *)
	fPositionAreaControlRange 		: LREAL;		(* 0x00000010 *)
	bEnableMotionControl			: WORD;		(* 0x00000011 *)
	fMotionControlTime 			: LREAL;		(* 0x00000012 *)
	bEnableLoop 				: WORD;		(* 0x00000013 *)
	fLoopDistance 				: LREAL;		(* 0x00000014 *)
	bEnableTargetPosControl 		: WORD;		(* 0x00000015 *)
	fTargetPosControlRange 		: LREAL;		(* 0x00000016 *)
	fTargetPosControlTime 		: LREAL;		(* 0x00000017 *)
	fVeloMaximum 				: LREAL;		(* 0x00000027 *)
	fMotionControlRange 			: LREAL;		(* 0x00000028 *)
	bEnablePEHTimeControl 		: WORD;		(* 0x00000029 *)
	fPEHControlTime 				: LREAL;		(* 0x0000002A *)
	bEnableBacklashCompensation : WORD;		(* 0x0000002B *)
	fBacklash 					: LREAL;		(* 0x0000002C *)
	sAmsNetId 					: T_AmsNetId;(* 0x00000031 (Wandlung von "BYTE b[6]" zum nullterminierten STRING mit 23+1 Zeichen) *)
	nPort 						: WORD;		(* 0x00000031 *)
	nChnNo 						: WORD;		(* 0x00000031 *)
	fAcceleration 					: LREAL;		(* 0x00000101 *)
	fDeceleration 					: LREAL;		(* 0x00000102 *)
	fJerk 						: LREAL;		(* 0x00000103 *)

	(* ENCODER: *)
	nEncId 						: DWORD;	(* 0x00010001 *)
	sEncName 					: STRING(31);	(* 0x00010002 *)
	nEncType 					: DWORD;	(* 0x00010003 *)
	fEncScaleFactor 				: LREAL;		(* 0x00010006 *)
	fEncOffset 					: LREAL;		(* 0x00010007 *)
	bEncIsInverse 				: WORD;		(* 0x00010008 *)
	fEncModuloFactor 			: LREAL;		(* 0x00010009 *)
	nEncMode 					: DWORD;	(* 0x0001000A *)
	bEncEnableSoftEndMinControl 	: WORD;		(* 0x0001000B *)
	bEncEnableSoftEndMaxControl 	: WORD;		(* 0x0001000C *)
	fEncSoftEndMin 				: LREAL;		(* 0x0001000D *)
	fEncSoftEndMax				: LREAL;		(* 0x0001000E *)
	nEncMaxIncrement 			: DWORD;	(* 0x00010015 *)
	bEncEnablePosCorrection 		: WORD;		(* 0x00010016 *)
	fEncPosCorrectionFilterTime 	: LREAL;		(* 0x00010017 *)

	(* CONTROLLER: *)
	nCtrlId 						: DWORD;	(* 0x00020001 *)
	sCtrlName 					: STRING(31);	(* 0x00020002 *)
	nCtrlType 					: DWORD;	(* 0x00020003 *)
	bCtrlEnablePosDiffControl 		: WORD;		(* 0x00020010 *)
	bCtrlEnableVeloDiffControl 		: WORD;		(* 0x00020011 *)
	fCtrlPosDiffMax				: LREAL;		(* 0x00020012 *)
	fCtrlPosDiffMaxTime 			: LREAL;		(* 0x00020013 *)
	fCtrlPosKp 					: LREAL;		(* 0x00020102 *)
	fCtrlPosTn 					: LREAL;		(* 0x00020103 *)
	fCtrlPosTv 					: LREAL;		(* 0x00020104 *)
	fCtrlPosTd 					: LREAL;		(* 0x00020105 *)
	fCtrlPosExtKp 					: LREAL;		(* 0x00020106 *)
	fCtrlPosExtVelo 				: LREAL;		(* 0x00020107 *)
	fCtrlAccKa 					: LREAL;		(* 0x00020108 *)

	(* DRIVE: *)
	nDriveId 						: DWORD;	(* 0x00030001 *)
	sDriveName 					: STRING(31);	(* 0x00030002 *)
	nDriveType 					: DWORD;	(* 0x00030003 *)
	bDriveIsInverse 				: WORD;		(* 0x00030006 *)
	fDriveVeloReferenz 			: LREAL;		(* 0x00030101 *)
	fDriveOutputReferenz 			: LREAL;		(* 0x00030102 *)

	(* fill up *)
	arrReserved : ARRAY[455..512] OF BYTE;		(* fill up to 512 bytes *)
END_STRUCT
END_TYPE

(* Data type *)
TYPE ST_AxisStatus :
STRUCT
	UpdateTaskIndex	: 	BYTE;	(* Task-Index of the task that updated this data set *)
	UpdateCycleTime	:	LREAL;	(* task cycle time of the task which calls the status function *)
	CycleCounter		: 	UDINT;	(* PLC cycle counter when this data set updated *)
	NcCycleCounter	: 	UDINT;	(* NC cycle counter incremented after NC task updated NcToPlc data structures *)

	MotionState 		: 	MC_AxisStates; 	(* motion state in the PLCopen state diagram *)

	Error			:	BOOL;	(* StateDWord bit 31 - axis error state *)
	ErrorID			:	UDINT;	(* axis error code *)

	(* PLCopen motion control statemachine states: *)
	ErrorStop		:	BOOL;
	Disabled			:	BOOL;
	Stopping			:	BOOL;
	StandStill		:	BOOL;
	DiscreteMotion	:	BOOL;
	ContinuousMotion	:	BOOL;	(* StateDWord bit 19 *)
	SynchronizedMotion:	BOOL;
	Homing			:	BOOL;

	(* additional status - (PLCopen definition)*)
	ConstantVelocity	:	BOOL;	(* StateDWord bit 12 *)
	Accelerating		:	BOOL;
	Decelerating		:	BOOL;

	(* Axis.NcToPlc.StateDWord *)
	Operational 		: 	BOOL;	(* StateDWord bit 0 - (was ready) *)
	ControlLoopClosed : 	BOOL;	(* StateDWord bit 20 - operational and position control active *)
	HasJob			: 	BOOL;	(* StateDWord bit 8 *)
	HasBeenStopped	: 	BOOL;	(* StateDWord bit 7 *)
	NewTargetPosition: 	BOOL;	(* StateDWord bit 17 - new target position commanded during move *)
	InPositionArea 	: 	BOOL;	(* StateDWord bit 3 *)
	InTargetPosition 	:	BOOL;	(* StateDWord bit 4 *)
(*	NotInTargetPosition:	BOOL;*)	(* StateDWord bit 18 - 20080610 KSt - not implemented*)
	Protected		:	BOOL;	(* StateDWord bit 5 *)
	Homed			: 	BOOL;	(* StateDWord bit 1 *)
	HomingBusy		: 	BOOL;	(* StateDWord bit 11 *)
	MotionCommandsLocked 	: BOOL; (* StateDWord bit 29 - stop 'n hold *)
	SoftLimitMinExceeded		: BOOL; (* StateDWord bit 26 - reverse soft travel limit exceeded *)
	SoftLimitMaxExceeded		: BOOL; (* StateDWord bit 27 - forward soft travel limit exceeded *)

	Moving			: 	BOOL;	(* StateDWord bit 9+10 *)
	PositiveDirection	: 	BOOL;	(* StateDWord bit 9 *)
	NegativeDirection : 	BOOL;	(* StateDWord bit 10 *)
	NotMoving		:	BOOL;	(* StateDWord bit 2 *)
	Compensating	: 	BOOL;	(* StateDWord bit 13 *) (* superposition - overlayed motion *)

	ExtSetPointGenEnabled : BOOL;	(* StateDWord bit 14 *)
	ExternalLatchValid	: 	BOOL;	(* StateDWord bit 16 *)
	CamDataQueued	: 	BOOL;	(* StateDWord bit 22 *)
	CamTableQueued :	BOOL;	(* StateDWord bit 21 *)
	CamScalingPending : 	BOOL;	(* StateDWord bit 23 *)
	CmdBuffered 		: 	BOOL;	(* StateDWord bit 24 *)
	PTPmode 		: 	BOOL;	(* StateDWord bit 25 *)
	DriveDeviceError	: 	BOOL;	(* StateDWord bit 28 *)
	IoDataInvalid 		: 	BOOL;	(* StateDWord bit 30 *)
	ErrorPropagationDelayed	: BOOL;	(* StateDWord bit 6 *)

	(* Axis.NcToPlc.CoupleState *)
	Coupled			: 	BOOL;

	(* axis operation mode feedback from NcToPlc *)
	OpMode			: 	ST_AxisOpModes;
END_STRUCT
END_TYPE

(* Data type *)
TYPE ST_DriveAddress :
STRUCT
	NetID			: T_AmsNetId;	(* AMS NetID of the drive as a string *)
	NetIdBytes		: T_AmsNetIdArr;	(* AMS NetID of the drive as a byte array (same information as NetID) *)
	SlaveAddress	: T_AmsPort;		(* slave address of the drive connected to a bus master *)
	Channel			: BYTE;			(* channel number of the drive *)
END_STRUCT
END_TYPE

(* Data type *)
TYPE ST_GearInDynOptions :
STRUCT
	CCVmode : BOOL; (* constant circumference velocity mode *)
END_STRUCT
END_TYPE

(* Data type *)
TYPE ST_GearInMultiMasterOptions :
STRUCT
	reserved : BOOL;
END_STRUCT
END_TYPE

(* Data type *)
TYPE ST_GearInOptions :
STRUCT
	SlaveType : _E_TcNC_SlaveTypes;
END_STRUCT
END_TYPE

(* Data type *)
TYPE ST_GearOutOptions :
STRUCT
	reserved : BOOL;
END_STRUCT
END_TYPE

(* Data type *)
TYPE ST_HomingOptions :
STRUCT
	ClearPositionLag 		: BOOL;	(* set actual and set position to same value and clear the position lag *)
END_STRUCT
END_TYPE

(* Data type *)
TYPE ST_McOutputs :
STRUCT
	Done				:	BOOL;
	Busy 				: 	BOOL;
	Active	 			: 	BOOL;
	CommandAborted		:	BOOL;
	Error				:	BOOL;
	ErrorID				:	UDINT;
END_STRUCT
END_TYPE

(* Data type *)
TYPE ST_MoveOptions :
STRUCT
	(* Command activation at defined ActivationPosition - extends the buffer mode when enabled *)
	EnableBlendingPosition : BOOL;
	BlendingPosition : LREAL;

	(* velocity profile options - instantaneous speed change at the beginning and at the end of the profile *)
	StartVelocity : LREAL;
	EndVelocity : LREAL;
END_STRUCT
END_TYPE

(* Data type *)
TYPE ST_PowerStepperStruct :
STRUCT
	DestallDetectMode	:	E_DestallDetectMode;
	DestallMode			:	E_DestallMode;
	DestallEnable		:	BOOL;
	StatusMonEnable		:	BOOL;

	Retries				:	INT;
	Timeout				:	TIME;
END_STRUCT
END_TYPE

(* Data type *)
TYPE ST_SetEncoderScalingOptions :
STRUCT
	SelectEncoderIndex 	: BOOL;	(* selects an encoder with index 0..n explicitly if enabled - selction by EncoderIndex below *)
	EncoderIndex 		: UINT;	(* encoder with index 0..n, 0 is first encoder - valid only if SelectEncoderIndex=TRUE *)
END_STRUCT
END_TYPE

(* Data type *)
TYPE ST_SetPositionOptions :
STRUCT
	ClearPositionLag 		: BOOL;	(* set actual and set position to same value and clear the position lag *)
	SelectEncoderIndex 	: BOOL;	(* selects an encoder with index 0..n explicitly if enabled - selction by EncoderIndex below *)
	EncoderIndex 		: UINT;	(* encoder with index 0..n, 0 is first encoder - valid only if SelectEncoderIndex=TRUE *)
END_STRUCT
END_TYPE

(* Data type *)
TYPE ST_SuperpositionOptions :
STRUCT
	AbortOption : E_SuperpositionAbortOption;
END_STRUCT
END_TYPE

(* Data type *)
TYPE ST_TableCharacValues :
STRUCT
    (* Master Velocity*)
	fMasterVeloNom	: LREAL;    (* 1.  master nominal velocity (normed: => 1.0) *)

	(* characteristic slave data *)
	(*===========================*)

   (* Start of cam table *)
	fMasterPosStart	: LREAL;	(* 2.  master start position *)
	fSlavePosStart	: LREAL;	(* 3.  slave start position *)
	fSlaveVeloStart	: LREAL;	(* 4.  slave start velocity *)
	fSlaveAccStart	: LREAL;	(* 5.  slave start acceleration *)
	fSlaveJerkStart	: LREAL;	(* 6.  slave start jerk *)

	(* End of cam table*)
	fMasterPosEnd	: LREAL;	(* 7.  master end position *)
	fSlavePosEnd	: LREAL;	(* 8.  slave end position *)
	fSlaveVeloEnd	: LREAL;	(* 9.  slave end velocity *)
	fSlaveAccEnd	: LREAL;	(* 10. slave end acceleration *)
	fSlaveJerkEnd	: LREAL;	(* 11. slave end jerk *)

	(* minimum slave position *)
	fMPosAtSPosMin	: LREAL;	(* 12. master position AT slave minimum position *)
	fSlavePosMin	: LREAL;	(* 13. slave minimum position *)

	(* minimum Slave velocity *)
	fMPosAtSVeloMin	: LREAL;	(* 14. master position AT slave minimum velocity *)
	fSlaveVeloMin	: LREAL;	(* 15. slave minimum velocity *)

	(* minimum slave acceleration *)
	fMPosAtSAccMin	: LREAL;	(* 16. master position AT slave minimum acceleration *)
	fSlaveAccMin	: LREAL;	(* 17. slave minimum acceleration *)
	fSVeloAtSAccMin	: LREAL;	(* 18. slave velocity AT slave minimum acceleration *)

	(* minimum slave jerk and dynamic momentum *)
	fSlaveJerkMin	: LREAL;	(* 19. slave minimum jerk *)
	fSlaveDynMomMin	: LREAL;	(* 20. slave minimum dynamic momentum (NOT SUPPORTED YET !) *)

	(* maximum slave position *)
	fMPosAtSPosMax	: LREAL;	(* 21. master position AT slave maximum position *)
	fSlavePosMax	: LREAL;	(* 22. slave maximum position *)

	(* maximum Slave velocity *)
	fMPosAtSVeloMax	: LREAL;	(* 23. master position AT slave maximum velocity *)
	fSlaveVeloMax	: LREAL;	(* 24. slave maximum velocity *)

	(* maximum slave acceleration *)
	fMPosAtSAccMax	: LREAL;	(* 25. master position AT slave maximum acceleration *)
	fSlaveAccMax	: LREAL;	(* 26. slave maximum acceleration *)
	fSVeloAtSAccMax	: LREAL;	(* 27. slave velocity AT slave maximum acceleration *)

	(* maximum Slave slave jerk and dynamic momentum *)
	fSlaveJerkMax	: LREAL;	(* 28. slave maximum jerk *)
	fSlaveDynMomMax	: LREAL;	(* 29. slave maximum dynamic momentum (NOT SUPPORTED YET !) *)

	(* mean and effective values *)
	fSlaveVeloMean	: LREAL;	(* 30. slave mean absolute velocity (NOT SUPPORTED YET !) *)
	fSlaveAccEff	: LREAL;	(* 31. slave effective acceleration (NOT SUPPORTED YET !) *)

	(* reserved space for future extension *)
	reserved 		: ARRAY[32..47] OF LREAL;

	(* organization structure of the cam table *)
	CamTableID 			: UDINT;
	NumberOfRows		: UDINT;	(* number of cam table entries, e. g. number of points *)
	NumberOfColumns	: UDINT;	(* number of table columns, typically 1 or 2 *)
	TableType			: INT;
	Periodic				: BOOL;

	reserved2 		: ARRAY[1..121] OF BYTE;
END_STRUCT
END_TYPE

(* Data type *)
TYPE TRIGGER_REF :
STRUCT
	EncoderID  	: UDINT;			(* 1..255 *)
	TouchProbe 	: E_TouchProbe;	(* Signal source *)
	Edge 		: E_SignalEdge;	(* rising or falling signal edge *)
	PlcEvent 	: BOOL;			(* PLC trigger signal input when TouchProbe signal source is set to 'PlcEvent' *)
	ModuloPositions : BOOL;		(* interpretation of FirstPosition, LastPosition and RecordedPosition as modulo positions when TRUE *)
	{library private}
	ProbeState 	: _E_TouchProbeState;	(* internal state of the touch probe sequence *)
END_STRUCT
END_TYPE

(* POU _F_AxisState, ST *)
{library private}
(* 	Function returns the current PLCopen axis state *)
(*	see state diagram *)
FUNCTION _F_AxisState : MC_AxisStates
VAR_IN_OUT
	NcToPlc : NCTOPLC_AXIS_REF;
	PlcToNc : PLCTONC_AXIS_REF;
END_VAR
VAR_INPUT
END_VAR
VAR
END_VAR
IF F_AxisInErrorState(NcToPlc.StateDWord) THEN
	IF PlcToNc.ControlDWord.0 THEN
		(* Power.Enable=TRUE but in error state *)
		_F_AxisState := MC_AXISSTATE_ERRORSTOP;
	ELSE
		_F_AxisState := MC_AXISSTATE_DISABLED;
	END_IF
ELSE
(*	IF F_AxisIsReady(NcToPlc.StateDWord) THEN *)			(* 20090205 KSt *)
	IF F_AxisControlLoopClosed(NcToPlc.StateDWord) THEN	(* 20090205 KSt *)
		IF F_AxisIsCoupled(NcToPlc.CoupleState) THEN
			(* slave *)
			_F_AxisState := MC_AXISSTATE_SYNCHRONIZEDMOTION;

		ELSIF F_AxisHasJob(NcToPlc.StateDWord) THEN
			(* moving single axis *)
			IF F_AxisHasBeenStopped(NcToPlc.StateDWord) THEN
				_F_AxisState := MC_AXISSTATE_STOPPING;
			ELSIF F_AxisIsCalibrating(NcToPlc.StateDWord) THEN
				_F_AxisState := MC_AXISSTATE_HOMING;
			ELSIF F_AxisIsMovingEndless(NcToPlc.StateDWord) THEN
				_F_AxisState := MC_AXISSTATE_CONTINOUSMOTION;
			ELSE
				_F_AxisState := MC_AXISSTATE_DISCRETEMOTION;
			END_IF
		ELSE
			(* ready but no job *)
			IF F_AxisMotionCommandsLocked(NcToPlc.StateDWord) THEN
				(* axis kept in stop mode by a stop command *)
				_F_AxisState := MC_AXISSTATE_STOPPING;
			ELSE
				_F_AxisState := MC_AXISSTATE_STANDSTILL;
			END_IF
		END_IF
	ELSE
		_F_AxisState := MC_AXISSTATE_DISABLED;
	END_IF
END_IF
END_FUNCTION

(* POU F_AxisInErrorState, ST *)
FUNCTION F_AxisInErrorState : BOOL
(* 	reference: 	NC -> PLC axis interface (128 bytes)
	check if bit 31 of an axis StateDWord is set:
	Axis is in a fault state
	Achse ist im Fehlerzustand
*)
VAR_INPUT
	StateDWord : DWORD;
END_VAR
VAR
END_VAR
F_AxisInErrorState := (StateDWord AND 2#1000_0000_0000_0000_0000_0000_0000_0000) <> 0;
END_FUNCTION

(* POU F_AxisControlLoopClosed, ST *)
FUNCTION F_AxisControlLoopClosed  : BOOL
(* 	reference: 	NC -> PLC axis interface (128 bytes)
	check if bit 20 of an axis StateDWord is set:
	Axis control loop is closed 
	Achsregelkreis ist geschlossen
*)
VAR_INPUT
	StateDWord : DWORD;
END_VAR
VAR
END_VAR
F_AxisControlLoopClosed := (StateDWord AND 2#0000_0000_0001_0000_0000_0000_0000_0000) <> 0;
END_FUNCTION

(* POU F_AxisIsCoupled, FBD *)
FUNCTION F_AxisIsCoupled : BOOL
VAR_INPUT
	nCoupleState : DWORD;
END_VAR
VAR
END_VAR
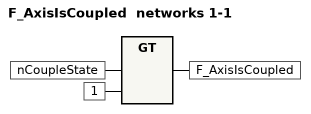
_FBD_ (* Function Block Diagram *)
NETWORK 1
	GT(nCoupleState, 1) => F_AxisIsCoupled
_END_FBD_
(* the same logic as Structured Text *)
(* Network 1 *)
F_AxisIsCoupled := nCoupleState > 1;
END_FUNCTION

(* POU F_AxisHasJob, ST *)
FUNCTION F_AxisHasJob : BOOL
(* 	reference: 	NC -> PLC axis interface (128 bytes)
	check if bit 8 of an axis StateDWord is set:
	Axis has instructions, is carrying instructions out
	Achse hat Auftrag, führt Auftrag aus
*)
VAR_INPUT
	StateDWord : DWORD;
END_VAR
VAR
END_VAR
F_AxisHasJob := (StateDWord AND 2#0000_0000_0000_0000_0000_0001_0000_0000) <> 0;
END_FUNCTION

(* POU F_AxisHasBeenStopped, ST *)
FUNCTION F_AxisHasBeenStopped : BOOL
(* 	reference: 	NC -> PLC axis interface (128 bytes)
	check if bit 7 of an axis StateDWord is set:
	Axis has been stopped or is presently executing a stop
	Achse ist gestoppt worden bzw. führt einen Stopp aus
*)
VAR_INPUT
	StateDWord : DWORD;
END_VAR
VAR
END_VAR
F_AxisHasBeenStopped := (StateDWord AND 2#0000_0000_0000_0000_0000_0000_1000_0000) <> 0;
END_FUNCTION

(* POU F_AxisIsCalibrating, ST *)
FUNCTION F_AxisIsCalibrating : BOOL
(* 	reference: 	NC -> PLC axis interface (128 bytes)
	check if bit 0 of an axis StateDWord is set:
	Axis is in referencing mode ("Axis being calibrated")
	Achse referenziert ("Achse wird geeicht")
*)
VAR_INPUT
	StateDWord : DWORD;
END_VAR
VAR
END_VAR
F_AxisIsCalibrating := (StateDWord AND 2#0000_0000_0000_0000_0000_1000_0000_0000) <> 0;
END_FUNCTION

(* POU F_AxisIsMovingEndless, ST *)
FUNCTION F_AxisIsMovingEndless  : BOOL
(* 	reference: 	NC -> PLC axis interface (128 bytes)
	check if bit 19 of an axis StateDWord is set:
	Axis is moving endless
	Achse in Endlos-Betriebsart
*)
VAR_INPUT
	StateDWord : DWORD;
END_VAR
VAR
END_VAR
F_AxisIsMovingEndless := (StateDWord AND 2#0000_0000_0000_1000_0000_0000_0000_0000) <> 0;
END_FUNCTION

(* POU F_AxisMotionCommandsLocked, ST *)
FUNCTION F_AxisMotionCommandsLocked : BOOL
(* 	reference: 	NC -> PLC axis interface (128 bytes)
	check if bit 29 of an axis StateDWord is set:
	Axis motion commands locked 
	Achse ist gegen Bewegungskommandos gesperrt 
*)
VAR_INPUT
	StateDWord : DWORD;
END_VAR
VAR
END_VAR
F_AxisMotionCommandsLocked := (StateDWord AND 2#0010_0000_0000_0000_0000_0000_0000_0000) <> 0;
END_FUNCTION

(* POU _F_GetIndexGroup, ST *)
{library private}
FUNCTION _F_GetIndexGroup : _ST_ParaStruct
VAR_INPUT
	ParaNumber	: INT;
	Mode		: INT; 		(* read/write *)
END_VAR
VAR
	IndexGroup	: UDINT;
	IndexOffset	: UDINT;
	nType 		: _E_ParameterType;
	lrValue		: LREAL;
END_VAR
(* set default values *)
_F_GetIndexGroup.IndexGroup 	:= 0;				(* default *)
_F_GetIndexGroup.IndexOffset 	:= 0;				(* default *)
_F_GetIndexGroup.ParaType 	:= PARAMETERTYPE_NOTYPE;	(* default *)
_F_GetIndexGroup.LrealSize	:= SIZEOF(lrValue);(* default *)
_F_GetIndexGroup.LrealOffset 	:= 1;				(* default *)
nType						:= PARAMETERTYPE_LREAL;	(* default *)
IndexOffset 					:= 0;				(* default *)
IndexGroup 					:= TcMcGlobal.Axis.Parameter.IDXGRP;	(* default *)

(* check parameter number and determine index group and index offset *)
CASE ParaNumber OF
(*				PLCopen specific parameters *)
(*				Beckhoff specific parameters *)
	AxisId 				:
		IndexOffset := 16#0000_0001;
		nType :=	PARAMETERTYPE_DWORD;
	AxisVeloManSlow :
		IndexOffset := 16#0000_0008;
	AxisVeloManFast :
		IndexOffset := 16#0000_0009;
	AxisVeloMax :
		IndexOffset := 16#0000_0027;
	AxisAcc, MaxAccelerationSystem, MaxAccelerationAppl 			:
		IndexOffset := 16#0000_0101;
	AxisDec, MaxDecelerationSystem, MaxDecelerationAppl 			:
		IndexOffset := 16#0000_0102;
	AxisJerk, MaxJerk 			:
		IndexOffset := 16#0000_0103;
	AxisMaxVelocity, MaxVelocitySystem, MaxVelocityAppl		:
		IndexOffset := 16#0000_0027;
	AxisRapidTraverseVelocity:
		IndexOffset := 16#0000_000A;
	AxisManualVelocityFast:
		IndexOffset := 16#0000_0009;
	AxisManualVelocitySlow:
		IndexOffset := 16#0000_0008;
	AxisCalibrationVelocityForward:
		IndexOffset := 16#0000_0006;
	AxisCalibrationVelocityBackward:
		IndexOffset := 16#0000_0007;
	AxisJogIncrementForward:
		IndexOffset := 16#0000_0018;
	AxisJogIncrementBackward:
		IndexOffset := 16#0000_0019;
	AxisMinSoftPosLimit, SWLimitNeg:
		IndexOffset := 16#0001_000D;
	AxisMaxSoftPosLimit, SWLimitPos:
		IndexOffset := 16#0001_000E;
	AxisMaxPosLagValue, MaxPositionLag:
		IndexOffset := 16#0002_0012;
	AxisMaxPosLagFilterTime:
		IndexOffset := 16#0002_0013;
	AxisPositionRangeWindow:
		IndexOffset := 16#0000_0010;
	AxisTargetPositionWindow:
		IndexOffset := 16#0000_0016;
	AxisTargetPositionMonitoringTime:
		IndexOffset := 16#0000_0017;
	AxisInTargetTimeout:
		IndexOffset := 16#0000_002A;
	AxisMotionMonitoringWindow:
		IndexOffset := 16#0000_0028;
	AxisMotionMonitoringTime:
		IndexOffset := 16#0000_0012;
	AxisDelayTimeVeloPosition:
		IndexOffset := 16#0000_0104;
	AxisLoopingDistance:
		IndexOffset := 16#0000_0014;
	AxisBacklash:
		IndexOffset := 16#0000_002C;
	AxisRefVeloOnRefOutput:
		IndexOffset := 16#0003_0101;
	AxisOverrideType:
		IndexOffset := 16#0000_0105;
		nType	:=  PARAMETERTYPE_DWORD;
	AxisEnMaxSoftPosLimit, EnableLimitPos:
		IndexOffset := 16#0001_000C;
		nType	:=  PARAMETERTYPE_BOOL;
	AxisEnMinSoftPosLimit, EnableLimitNeg:
		IndexOffset := 16#0001_000B;
		nType	:=  PARAMETERTYPE_BOOL;
	AxisEnPositionLagMonitoring, EnablePosLagMonitoring:
		IndexOffset := 16#0002_0010; (* 4.12.03 KSt, change 0002_0012 to 0002_0010 *)
		nType	:=  PARAMETERTYPE_BOOL;
	AxisEnPositionRangeMonitoring:
		IndexOffset := 16#0000_000F;
		nType	:=  PARAMETERTYPE_BOOL;
	AxisEnTargetPositionMonitoring:
		IndexOffset := 16#0000_0015;
		nType	:=  PARAMETERTYPE_BOOL;
	AxisEnInTargetTimeout:
		IndexOffset := 16#0000_0029;
		nType	:=  PARAMETERTYPE_BOOL;
	AxisEnMotionMonitoring:
		IndexOffset := 16#0000_0011;
		nType	:=  PARAMETERTYPE_BOOL;
	AxisEnLoopingDistance:
		IndexOffset := 16#0000_0013;
		nType	:=  PARAMETERTYPE_BOOL;
	AxisEnBacklashCompensation:
		IndexOffset := 16#0000_002B;
		nType	:=  PARAMETERTYPE_BOOL;
	AxisEnDataPersistence:
		IndexOffset := 16#0000_0030;
		nType	:=  PARAMETERTYPE_BOOL;
	AxisEncoderScalingFactor :
		IndexOffset := 16#0001_0006;
	AxisEncoderOffset :
		IndexOffset := 16#0001_0007;
	AxisEncoderDirectionInverse :
		IndexOffset := 16#0001_0008;
		nType	:=  PARAMETERTYPE_BOOL;
	AxisEncoderMask :
		IndexOffset := 16#0001_0015;
		nType	:=  PARAMETERTYPE_DWORD;
	AxisEncoderModuloValue :
		IndexOffset := 16#0001_0009;
	AxisModuloToleranceWindow :
		IndexOffset := 16#0001_001B;
	AxisEnablePosCorrection :
		IndexOffset := 16#0001_0016;
		nType	:=  PARAMETERTYPE_BOOL;
	AxisPosCorrectionFilterTime :
		IndexOffset := 16#0001_0017;
	AxisUnitInterpretation :	(* added 5/20/2008 KSt *)
		IndexOffset := 16#0000_0026;
		nType	:= PARAMETERTYPE_DWORD;
	AxisMotorDirectionInverse :	(* added 1/11/2010 KSt *)
		IndexOffset := 16#0003_0006;
		nType	:=  PARAMETERTYPE_BOOL;

	(* check for status information *)
	AxisTargetPosition:
		IndexGroup := TcMcGlobal.Axis.State.IDXGRP;
		IndexOffset := 16#0000_0013;
	AxisRemainingTimeToGo:
		IndexGroup := TcMcGlobal.Axis.State.IDXGRP;
		IndexOffset := 16#0000_0014;
		_F_GetIndexGroup.LrealSize := 2 * SIZEOF(lrValue);	(* read data structure with two lreal values *)
		_F_GetIndexGroup.LrealOffset := 1;	(* get first lreal value *)
	AxisRemainingDistanceToGo:
		IndexGroup := TcMcGlobal.Axis.State.IDXGRP;
		IndexOffset := 16#0000_0014;
		_F_GetIndexGroup.LrealSize := 2 * SIZEOF(lrValue);	(* read data structure with two lreal values *)
		_F_GetIndexGroup.LrealOffset := 2;	(* get second lreal value *)

	(* check for axis function information *)
	AxisGearRatio:
		(* gear ratio is status information in read mode but a function call in write mode *)
		IndexGroup := SEL( Mode=READWRITEPARAMETERMODE_WRITE, TcMcGlobal.Axis.State.IDXGRP, TcMcGlobal.Axis.Functions.IDXGRP );
		IndexOffset := SEL(Mode=READWRITEPARAMETERMODE_WRITE, 16#0000_0022, 16#0000_0042 );
		_F_GetIndexGroup.LrealSize := 4 * SIZEOF(lrValue);	(* read data structure with four lreal values *)
		_F_GetIndexGroup.LrealOffset := 1;	(* get first lreal value *)
ELSE
	nType		:=  PARAMETERTYPE_NOTYPE;	(* not found *)
END_CASE;

IF IndexOffset <> 0 THEN
	_F_GetIndexGroup.IndexGroup := IndexGroup;
	_F_GetIndexGroup.IndexOffset := IndexOffset;
	_F_GetIndexGroup.ParaType := nType;
END_IF
END_FUNCTION

(* POU _F_ReadStatus, ST *)
{library private}
FUNCTION _F_ReadStatus : ST_AxisStatus
VAR_IN_OUT
	NcToPlc : NCTOPLC_AXIS_REF;
	PlcToNc : PLCTONC_AXIS_REF;
END_VAR
VAR
	GetTaskIndex : GETCURTASKINDEX;
END_VAR
 (* MOTION CONTROL STATEMACHINE STATES *)
_F_ReadStatus.ErrorStop			:= FALSE;
_F_ReadStatus.Disabled 			:= FALSE;
_F_ReadStatus.Stopping			:= FALSE;
_F_ReadStatus.StandStill			:= FALSE;
_F_ReadStatus.DiscreteMotion		:= FALSE;
_F_ReadStatus.ContinuousMotion	:= FALSE;
_F_ReadStatus.SynchronizedMotion	:= FALSE;
_F_ReadStatus.Homing			:= FALSE;

_F_ReadStatus.MotionState := _F_AxisState(NcToPlc, PlcToNc);
CASE _F_ReadStatus.MotionState OF
	MC_AXISSTATE_DISABLED :
		_F_ReadStatus.Disabled := TRUE;
	MC_AXISSTATE_STANDSTILL :
		_F_ReadStatus.StandStill := TRUE;
	MC_AXISSTATE_ERRORSTOP :
		_F_ReadStatus.ErrorStop := TRUE;
	MC_AXISSTATE_STOPPING :
		_F_ReadStatus.Stopping := TRUE;
	MC_AXISSTATE_HOMING :
		_F_ReadStatus.Homing	:= TRUE;
	MC_AXISSTATE_DISCRETEMOTION :
		_F_ReadStatus.DiscreteMotion := TRUE;
	MC_AXISSTATE_CONTINOUSMOTION :
		_F_ReadStatus.ContinuousMotion := TRUE;
	MC_AXISSTATE_SYNCHRONIZEDMOTION :
		_F_ReadStatus.SynchronizedMotion := TRUE;
END_CASE

(* NcToPlc.StateDWord *)
_F_ReadStatus.Operational				:= NcToPlc.StateDWord.0;
_F_ReadStatus.Homed				:= NcToPlc.StateDWord.1;		(* homed *)
_F_ReadStatus.NotMoving				:= NcToPlc.StateDWord.2;
_F_ReadStatus.InPositionArea			:= NcToPlc.StateDWord.3;
_F_ReadStatus.inTargetPosition 		:= NcToPlc.StateDWord.4;
_F_ReadStatus.Protected				:= NcToPlc.StateDWord.5;
_F_ReadStatus.ErrorPropagationDelayed	:= NcToPlc.StateDWord.6;
_F_ReadStatus.HasBeenStopped		:= NcToPlc.StateDWord.7;
_F_ReadStatus.HasJob				:= NcToPlc.StateDWord.8;
_F_ReadStatus.Moving				:= NcToPlc.StateDWord.9 OR NcToPlc.StateDWord.10;
_F_ReadStatus.PositiveDirection		:= NcToPlc.StateDWord.9;
_F_ReadStatus.NegativeDirection 		:= NcToPlc.StateDWord.10;
_F_ReadStatus.HomingBusy			:= NcToPlc.StateDWord.11; 	(* homing *)
_F_ReadStatus.ConstantVelocity 		:= NcToPlc.StateDWord.12;
_F_ReadStatus.Compensating			:= NcToPlc.StateDWord.13;	(* superposition active *)
_F_ReadStatus.ExtSetPointGenEnabled 	:= NcToPlc.StateDWord.14;
(* 15  busy *)
_F_ReadStatus.ExternalLatchValid		:= NcToPlc.StateDWord.16;
_F_ReadStatus.NewTargetPosition		:= NcToPlc.StateDWord.17;
(*_F_ReadStatus.NotInTargetPosition 	:= NcToPlc.StateDWord.18; 20080610 KSt  - not implemented *)
(*_F_ReadStatus.MovingEndless 		:= NcToPlc.StateDWord.19;	see continuous motion *)
_F_ReadStatus.ControlLoopClosed 		:= NcToPlc.StateDWord.20;
_F_ReadStatus.CamTableQueued 		:= NcToPlc.StateDWord.21;
_F_ReadStatus.CamDataQueued		:= NcToPlc.StateDWord.22;
_F_ReadStatus.CamScalingPending 		:= NcToPlc.StateDWord.23;
_F_ReadStatus.CmdBuffered	 		:= NcToPlc.StateDWord.24;
_F_ReadStatus.PTPmode	 			:= NcToPlc.StateDWord.25;
_F_ReadStatus.SoftLimitMinExceeded	:= NcToPlc.StateDWord.26;
_F_ReadStatus.SoftLimitMaxExceeded	:= NcToPlc.StateDWord.27;
_F_ReadStatus.DriveDeviceError	 	:= NcToPlc.StateDWord.28;
_F_ReadStatus.MotionCommandsLocked	:= NcToPlc.StateDWord.29;
_F_ReadStatus.IoDataInvalid			:= NcToPlc.StateDWord.30;
_F_ReadStatus.Error 					:= NcToPlc.StateDWord.31;

(* NcToPlc.nCoupleState *)
_F_ReadStatus.Coupled		:= NcToPlc.CoupleState > 1;

(* additional status data structue *)
_F_ReadStatus.ErrorID			:= NcToPlc.ErrorCode;
_F_ReadStatus.Accelerating 	:= NcToPlc.AxisState = TCNC_PHASE_ACCPOS;
_F_ReadStatus.Decelerating 	:= NcToPlc.AxisState = TCNC_PHASE_ACCNEG;

(* axis operation modes *)
_F_ReadStatus.OpMode.PositionAreaMonitoring	:= NcToPlc.OpModeDWord.0;
_F_ReadStatus.OpMode.TargetPositionMonitoring	:= NcToPlc.OpModeDWord.1;
_F_ReadStatus.OpMode.LoopMode				:= NcToPlc.OpModeDWord.2;
_F_ReadStatus.OpMode.MotionMonitoring		:= NcToPlc.OpModeDWord.3;
_F_ReadStatus.OpMode.PEHTimeMonitoring		:= NcToPlc.OpModeDWord.4;
_F_ReadStatus.OpMode.BacklashCompensation	:= NcToPlc.OpModeDWord.5;
_F_ReadStatus.OpMode.DelayedErrorReaction	:= NcToPlc.OpModeDWord.6;	(* 2008-02-20 KSt *)
_F_ReadStatus.OpMode.Modulo				:= NcToPlc.OpModeDWord.7;
_F_ReadStatus.OpMode.PositionLagMonitoring	:= NcToPlc.OpModeDWord.16;
_F_ReadStatus.OpMode.VelocityLagMonitoring	:= NcToPlc.OpModeDWord.17;
_F_ReadStatus.OpMode.SoftLimitMinMonitoring	:= NcToPlc.OpModeDWord.18;
_F_ReadStatus.OpMode.SoftLimitMaxMonitoring	:= NcToPlc.OpModeDWord.19;
_F_ReadStatus.OpMode.PositionCorrection		:= NcToPlc.OpModeDWord.20;
_F_ReadStatus.OpMode.AllowSlaveCommands	:= NcToPlc.OpModeDWord.21;	(* 2008-02-20 KSt *)

(* NC cycle counter will be incremented after NC task updated the NcToPlc data structure *)
_F_ReadStatus.NcCycleCounter := SHR(NcToPlc.OpModeDWord, 24);

GetTaskIndex();
_F_ReadStatus.UpdateTaskIndex := GetTaskIndex.index;
_F_ReadStatus.CycleCounter := SystemTaskInfoArr[_F_ReadStatus.UpdateTaskIndex].cycleCount;
_F_ReadStatus.UpdateCycleTime := SystemTaskInfoArr[_F_ReadStatus.UpdateTaskIndex].cycleTime / 1.0E6;	(* Correction 2009-11-26 KSt *)
(*
IF SystemTaskInfoArr[_F_ReadStatus.UpdateTaskIndex].cycleTime > 0 THEN
	_F_ReadStatus.UpdateCycleTime := 1000.0 / SystemTaskInfoArr[_F_ReadStatus.UpdateTaskIndex].cycleTime;
END_IF
*)
END_FUNCTION

(* POU _F_TcMC_DWORD_TO_HEXSTR, ST *)
{library private}
FUNCTION _F_TcMC_DWORD_TO_HEXSTR : STRING(4)
(* convert a decimal number to a hex string *)
VAR_INPUT
	in				: DWORD;
END_VAR
VAR
	str1 : STRING(4);
	pstr: POINTER TO BYTE;
	i: INT;
	digit: BYTE;
END_VAR
str1 := '@@@@';
pstr := ADR(str1) + 4;
FOR i := 1 TO 4 DO
	pstr := pstr - 1;
	digit := DWORD_TO_BYTE(in AND 16#F);
	IF digit < 10 THEN
		digit := digit + 48;
	ELSE
		digit := digit + 65 - 10;
	END_IF
	pstr^ := digit;
	in := in / 16;
END_FOR
_F_TcMC_DWORD_TO_HEXSTR := str1;
END_FUNCTION

(* POU _F_TcMC_Round, ST *)
{library private}
FUNCTION _F_TcMC_Round : LREAL
VAR_INPUT
	value : LREAL;
	digits : BYTE;
END_VAR
VAR
	n: LREAL;
END_VAR
n := EXPT(10, digits);
_F_TcMC_Round := FLOOR(value*n+0.5)/n;
END_FUNCTION

(* POU _FB_MoveUniversalGeneric, ST *)
FUNCTION_BLOCK _FB_MoveUniversalGeneric
VAR_IN_OUT
	Axis				:	AXIS_REF;
	LastExecutionResult: _ST_FunctionBlockResults;
END_VAR
VAR_INPUT
	Execute			:	BOOL;
	StartType		: 	UDINT;
	Position			:	LREAL;
	Velocity			:	LREAL;
	Acceleration		:	LREAL;
	Deceleration		:	LREAL;
	Jerk				:	LREAL;
(*	Direction			:	MC_Direction := MC_Positive_Direction;	*)(* E *)
	BufferMode		:	MC_BufferMode;
	Options			: 	ST_MoveOptions;
	Reset			: 	BOOL;	(* for internal use only *)
	GotoRunState	: 	BOOL;	(* for internal use only *)
END_VAR
VAR_OUTPUT
	Done				:	BOOL;	(* Same meaning as InVelocity for continous motion commands *)
	Busy 				: 	BOOL;
	Active	 			: 	BOOL;
	CommandAborted		:	BOOL;
	Error				:	BOOL;
	ErrorID				:	UDINT;
	CmdNo				: 	UINT;
	ADSbusy: BOOL;
END_VAR
VAR
	iState			: 	_E_TcMC_STATES := STATE_INITIALIZATION;
	sStartRequest	:	_ST_TcNC_UnversalAxisStartRequest;
	sStartResponse	:	_ST_TcNC_UnversalAxisStartResponse;
	fbAdsReadWrite	: 	ADSRDWRTEX;
	ContinousMode	: 	BOOL;
	InVelocity		: 	BOOL;
END_VAR
{library private}
VAR
	EmptyStartResponse	: 	_ST_TcNC_UnversalAxisStartResponse;
	COUNT_R			: 	UDINT;
	CounterCmdNoZero	: 	BYTE;
	CounterCmdNotStarted	: 	BYTE;
	NcCycleCounter		:	BYTE;
	LastNcCycleCounter	:	BYTE;
	NcMappingCounter 	: 	BYTE;
	NcCycleCounterAvailable: 	BOOL;
	NcCycleCounterNotAvailable: 	BOOL;
	NcCyclicFeedbackExpected: BOOL;
	PlcDebugCode 		: 	DWORD;	(* additional information for debugging purposes will be added to debug messages (ActErrorMessage) *)
	AxisIsSlave			: 	BOOL;
	fbTimeOut			:	TON;
	fbOnTrigger			:	R_TRIG;
	sTempMsg			: 	STRING(255);
END_VAR
VAR CONSTANT
	OpMode : _ST_TcNc_OperationModes;
END_VAR
(* ====================================================================== *)
(* *)
(* ====================================================================== *)
IF Reset THEN
	(* Reset FB for internal use only *)
	InVelocity := FALSE;
	Done := FALSE;
	Busy := FALSE;
	Active := FALSE;
	CommandAborted := FALSE;
	Error := FALSE;
	ErrorID := 0;
	fbAdsReadWrite( WRTRD := FALSE );
	iState := STATE_INITIALIZATION;
END_IF

fbOnTrigger(CLK:= Execute);

CASE iState OF
STATE_INITIALIZATION:	(* *)
	Busy := FALSE;
	Active := FALSE;
	IF NOT Execute THEN
		Done := FALSE;
		CommandAborted := FALSE;
		Error := FALSE;			(* reset at falling edge of Execute *)
		ErrorID := 0;
	END_IF
    	IF fbOnTrigger.Q THEN
		(* initialize output values *)
		Done := FALSE;
		InVelocity := FALSE;
		Busy := TRUE;
		Active := FALSE;
		CommandAborted := FALSE;
		Error := FALSE;
		ErrorID := 0;
		NcCyclicFeedbackExpected := FALSE;
		LastExecutionResult.Done := FALSE;
		LastExecutionResult.CommandAborted := FALSE;
		LastExecutionResult.Error := FALSE;
		LastExecutionResult.ErrorID := 0;
		CounterCmdNoZero := 0;
		CounterCmdNotStarted := 0;
		PlcDebugCode := Axis.PlcToNc.Reserved1;	(* additional information for debugging purposes will be added to debug messages (ActErrorMessage) *)
		(* nCmdNo := 0; *)
		fbTimeOut(IN:= FALSE);
		fbAdsReadWrite(WRTRD:=FALSE);

		IF GotoRunState THEN
			(* reset mapping counter *)
			NcMappingCounter := 0;
			LastNcCycleCounter:=DWORD_TO_BYTE(SHR(Axis.NcToPlc.OpModeDWord, 24));
			NcCyclicFeedbackExpected := FALSE;
			ActNcCycleCounter;
			iState := STATE_RUNNING;
		ELSE
			IF	NOT Axis.NcToPlc.StateDWord.6 (* error delay mode - pass any command during error delay - 2008-11-26 KSt *)
				AND StartType <> TCNC_START_STOPANDLOCK (* no pre-checks for stop and halt - 2008-11-26 KSt *)
				AND StartType<> TCNC_START_HALT (* no pre-checks for stop and halt - 2008-11-26 KSt *)
				THEN
				(* check for error conditions that don't allow to pass a command *)
				IF F_AxisInErrorState(Axis.NcToPlc.StateDWord) THEN
					Error := TRUE;
					ErrorID := Axis.NcToPlc.ErrorCode;
				ELSIF F_AxisInProtectedMode(Axis.NcToPlc.StateDWord) AND ((Axis.NcToPlc.OpModeDWord AND OpMode.AllowSlaveCommands) = 0) THEN (* 2008-02-20 KSt *)
(*				ELSIF F_AxisInProtectedMode(Axis.NcToPlc.StateDWord) THEN *)	 (* 2008-02-20 KSt *)
					(* motion commands on slaves not allowed *)
					Error := TRUE;
					ErrorID := MC_ERROR_AXIS_IN_PROTECTED_MODE;
				ELSIF NOT F_AxisIsReady(Axis.NcToPlc.StateDWord) THEN
					Error := TRUE;
					ErrorID := MC_ERROR_AXIS_IS_NOT_READY;
				ELSIF StartType = 0 THEN
					Error := TRUE;
					ErrorID := MC_ERROR_COMMAND_NOT_ALLOWED;
				END_IF
			END_IF
			IF NOT Error THEN (* pass the command to the NC *)
				(* universal axis start *)
				(* fill struct *)
				CASE StartType OF
					TCNC_START_ENDLESS_PLUS,
					TCNC_START_ENDLESS_MINUS,
					TCNC_START_ENDLESSPLUS_SLOWMANUAL,
					TCNC_START_ENDLESSMINUS_SLOWMANUAL,
					TCNC_START_ENDLESSPLUS_FASTMANUAL,
					TCNC_START_ENDLESSMINUS_FASTMANUAL:
						ContinousMode := TRUE;
					ELSE
						ContinousMode := FALSE;
				END_CASE
				AxisIsSlave := F_AxisIsCoupled(Axis.NcToPlc.CoupleState);
				sStartRequest.nStartType := StartType;
				sStartRequest.nControlMask := SEL(Options.EnableBlendingPosition, 0, 1);
				sStartRequest.fPosTarget := Position;
				sStartRequest.fVeloRequ := Velocity;
				sStartRequest.fAcc := Acceleration;
				sStartRequest.fDec := Deceleration;
				sStartRequest.fJerk := Jerk;
				sStartRequest.nBufferMode := BufferMode;
				sStartRequest.fBlendingPosition := Options.BlendingPosition;
				sStartRequest.fVeloStart := Options.StartVelocity;
				sStartRequest.fVeloEnd := Options.EndVelocity;
				sStartResponse := EmptyStartResponse;

				fbAdsReadWrite.PORT := SEL(AxisIsSlave, AMSPORT_R0_NCSAF, TcMcGlobal.NCPORT_TCMC_COUPLING); (* select SAF port or standard port when coupled *)
				fbAdsReadWrite.PORT := SEL(Axis.ADS.Port = 0, Axis.ADS.port, fbAdsReadWrite.PORT); (* override with user defined port *)
				fbAdsReadWrite.IDXOFFS := SEL(AxisIsSlave,
								TcMcGlobal.Axis.Functions.IDXOFFS.UNIVERSALSTART,			(* standalone axes *)
								TcMcGlobal.Axis.Functions.IDXOFFS.SLAVEUNIVERSALSTART);	(* slave axes with automatic decoupling *)
				fbAdsReadWrite(
					NETID:= Axis.ADS.netId,
					IDXGRP:= TcMcGlobal.Axis.Functions.IDXGRP + Axis.NcToPlc.AxisId,
					(* IDXOFFS:= TcMcGlobal.Axis.Functions.IDXOFFS.UNIVERSALSTART, *) (* 24.2.09 KSt - see offset selection above *)
					WRITELEN:= SIZEOF(sStartRequest),
					READLEN:= SIZEOF(sStartResponse),
					SRCADDR:= ADR(sStartRequest),
					DESTADDR:= ADR(sStartResponse),
					WRTRD:= TRUE,
					TMOUT:= TcMcGlobal.tADSTimeOut,
					COUNT_R=> COUNT_R );

				iState := STATE_ORDER;
			END_IF;
		END_IF;
	END_IF;

STATE_ORDER:  (* wait until command is accepted *)
	fbAdsReadWrite(COUNT_R=> COUNT_R );
	IF NOT fbAdsReadWrite.Busy THEN
		IF fbAdsReadWrite.Err OR COUNT_R <> SIZEOF(sStartResponse) THEN
			Error := TRUE;
			ErrorID := fbAdsReadWrite.ErrId;
			ActErrorMessage;
			iState := STATE_INITIALIZATION;
		ELSE
			CmdNo := sStartResponse.nCmdNo;
			Active := CmdNo = Axis.NcToPlc.CmdNo;
(*			ActErrorMessage; *)
			(* reset mapping counter *)
			NcMappingCounter := 0;
			LastNcCycleCounter:=DWORD_TO_BYTE(SHR(Axis.NcToPlc.OpModeDWord, 24));
			NcCyclicFeedbackExpected := FALSE;
			ActNcCycleCounter;

			iState := STATE_RUNNING;
		END_IF
	END_IF

STATE_RUNNING:  (* wait until axis stands still *)
	ActNcCycleCounter;
	Active := sStartResponse.nCmdNo = Axis.NcToPlc.CmdNo;
	IF Active THEN
		(* command is active and the axis motion status must be monitored *)
		IF (StartType=TCNC_START_STOPANDLOCK) OR (StartType=TCNC_START_HALT) THEN
			ActMonitorStop; 			(* used with MC_Halt and MC_Stop *)
		ELSIF ContinousMode THEN
			ActMonitorContinousMotion; (* used with e. g. MoveVelocity *)
		ELSE
			ActMonitorDiscreteMotion;	(* used with e. g. MoveAbsolute *)
		END_IF

	ELSE (* command not yet active *)
		IF F_AxisIsCoupled(Axis.NcToPlc.CoupleState) THEN	(* 20090205 KSt *)
			(* if axis is coupled during motion (FlyingSaw) all commands are aborted - 20090205 KSt*)
			CommandAborted := TRUE;
			iState := STATE_INITIALIZATION;
		ELSIF Axis.NcToPlc.CmdNo = 0 AND NcCyclicFeedbackExpected THEN  				(* 20090206 KSt *)
			CounterCmdNoZero := CounterCmdNoZero + 1;
			IF CounterCmdNoZero > TcMcGlobal.NCTOPLC_FEEDBACK_MAXWAITCYCLES THEN (* wait for a certain number of cycles before error *)
				(* CmdNo zero is not supposed to happen - it may come up after a coupling situation for a few cycles *)
				Error := TRUE;
				ErrorID := MC_ERROR_BUFFERED_COMMAND_CMDNOZERO; (* no command state feedback from NC *)
				iState := STATE_INITIALIZATION;
			END_IF
		ELSIF Axis.NcToPlc.CmdNo = (sStartResponse.nCmdNo + 1) OR
		     	((Axis.NcToPlc.CmdNo = 1) AND  (sStartResponse.nCmdNo=16#FFFF)) (* overrun with a difference of 1 *)
			THEN
			(* feedback CmdNo is exactly ONE increment higher than my command *)
			(* command was aborted or successfully finished *)
			Error := GETBIT32(Axis.NcToPlc.CmdState, INT_TO_SINT(CMDSTATE_LASTCMD_ENDED_WITH_ERROR));
			CommandAborted := NOT Error AND GETBIT32(Axis.NcToPlc.CmdState, INT_TO_SINT(CMDSTATE_LASTCMD_ABORTED_WITHOUT_ERROR));
			Done := NOT Error AND NOT Done AND GETBIT32(Axis.NcToPlc.CmdState, INT_TO_SINT(CMDSTATE_LASTCMD_SUCCESSFULLY_EXECUTED));
			IF Error THEN
				(* if axis error-Id is valid then feed it back - otherwhise errror-Id is unknown. *)
				ErrorID := SEL(Axis.NcToPlc.ErrorCode=0, Axis.NcToPlc.ErrorCode, MC_ERROR_BUFFERED_COMMAND_ERRORID_NOT_AVAILABLE  );
			END_IF
			IF NOT Done AND NOT CommandAborted AND NOT Error THEN
				Error := TRUE;
				ErrorID := MC_ERROR_BUFFERED_COMMAND_NO_STATE_FEEDBACK; (* no command state feedback from NC *)
			END_IF
			iState := STATE_INITIALIZATION;
		ELSIF Axis.NcToPlc.CmdNo = (sStartResponse.nCmdNo + 2) OR
		     	((Axis.NcToPlc.CmdNo = 2) AND  (sStartResponse.nCmdNo=16#FFFF)) (* overrun with a difference of 1 *)
			THEN
			(* feedback CmdNo is exactly TWO increments higher than my command  - 20090116 KSt *)
			Error := GETBIT32(Axis.NcToPlc.CmdState, INT_TO_SINT(CMDSTATE_LASTCMD_ENDED_WITH_ERROR)); (* error of command+1 *)
			(* if command+1 was aborted then this command has been aborted as well *)
			CommandAborted := NOT Error AND GETBIT32(Axis.NcToPlc.CmdState, INT_TO_SINT(CMDSTATE_LASTCMD_ABORTED_WITHOUT_ERROR));
			IF NOT CommandAborted THEN
				(* if previous command has not been aborted - the status of this command is unknown *)
				Error := TRUE;
				ErrorID := MC_ERROR_BUFFERED_COMMAND_MONITORING_IMPOSSIBLE; (* additional error code with command aborted *)
			END_IF
			iState := STATE_INITIALIZATION;
		 ELSIF 	Axis.NcToPlc.CmdNo > sStartResponse.nCmdNo OR
		     	((Axis.NcToPlc.CmdNo < 16#4000) AND  (sStartResponse.nCmdNo>16#A000)) (* overrun *)
			THEN
			(* feedback CmdNo is THREE or more increments higher than my command *)
			(* command was aborted - command monitoring impossible *)
			Error := TRUE;
			ErrorID := MC_ERROR_BUFFERED_COMMAND_MONITORING_IMPOSSIBLE; (* additional error code with command aborted *)
			(*CommandAborted := TRUE;*)	(*  20090116 KSt *)
			iState := STATE_INITIALIZATION;
		ELSIF F_AxisInErrorState(Axis.NcToPlc.StateDWord) THEN
			(* axis error came up before this command has been started *)
			Error := TRUE;
			ErrorID := AXIS.NcToPlc.ErrorCode;
			iState := STATE_INITIALIZATION;
		ELSIF NOT F_AxisHasJob(Axis.NcToPlc.StateDWord) AND NcCyclicFeedbackExpected THEN
			(* CmdNo is still lower than my command - command has not been initiated *)
			IF F_AxisHasBeenStopped(Axis.NcToPlc.StateDWord) THEN
				CommandAborted := TRUE;		(* stopp command aborts this command *)
				iState := STATE_INITIALIZATION;
			ELSE
				(* other cases are not supposed to happen and are error conditions *)
				CounterCmdNotStarted := CounterCmdNotStarted + 1;
				IF CounterCmdNotStarted > TcMcGlobal.NCTOPLC_FEEDBACK_MAXWAITCYCLES THEN (* wait for a certain number of cycles before error *)
					Error := TRUE;
					ErrorID := MC_ERROR_BUFFERED_COMMAND_NOT_STARTED; (* reason unknown *)
					iState := STATE_INITIALIZATION;
				END_IF
			END_IF
			(* timeout check *);
		END_IF
	END_IF
	IF (Error OR CommandAborted) AND (iState<>STATE_RUNNING) THEN
		ActErrorMessage;
	END_IF

ELSE  (* CASE : Unknown program state *)
	iState:= STATE_INITIALIZATION;
END_CASE

ADSbusy := fbAdsReadWrite.BUSY;
IF iState=STATE_INITIALIZATION THEN
	(* reset Busy immediately  when sequence ends *)
	IF Busy THEN
		LastExecutionResult.Done := Done;
		LastExecutionResult.CommandAborted := CommandAborted;
		LastExecutionResult.Error := Error;
		LastExecutionResult.ErrorID := ErrorID;
	END_IF
	Busy := FALSE;
	Active := FALSE;
END_IF
END_FUNCTION_BLOCK
ACTION ActErrorMessage:
IF Axis.PlcToNc.ControlDWord.30 THEN (* bit 30 - debug mode enabled *)
	(* FEHLERMELDUNG *)
	sTempMsg	:= 'TCMC:UAS Axis '; 	(* UAS = universal axis start *)
	sTempMsg	:= CONCAT( sTempMsg, UDINT_TO_STRING( Axis.NcToPlc.AxisId ) );
	sTempMsg	:= CONCAT( sTempMsg, ', CmdNo: ' );
	sTempMsg	:= CONCAT( sTempMsg, UDINT_TO_STRING( sStartResponse.nCmdNo ) );
	IF Error THEN
		sTempMsg	:= CONCAT( sTempMsg, ', Error: 0x' );
		sTempMsg	:= CONCAT( sTempMsg, _F_TcMC_DWORD_TO_HEXSTR(ErrorID) );
	END_IF
	IF CommandAborted THEN
		sTempMsg	:= CONCAT( sTempMsg, ', ABORTED ' );
	END_IF
	sTempMsg	:= CONCAT( sTempMsg, ', StartType: ' );
	sTempMsg	:= CONCAT( sTempMsg, UDINT_TO_STRING( sStartRequest.nStartType ) );
	sTempMsg	:= CONCAT( sTempMsg, ', SetPos: ' );
	sTempMsg	:= CONCAT( sTempMsg, LREAL_TO_STRING( _F_TcMC_Round( Axis.NcToPlc.SetPos , 4) ) );
	sTempMsg	:= CONCAT( sTempMsg, ', SetVelo: ' );
	sTempMsg	:= CONCAT( sTempMsg, LREAL_TO_STRING( _F_TcMC_Round( Axis.NcToPlc.SetVelo, 4) ) );
	sTempMsg	:= CONCAT( sTempMsg, ', SetAcc: ' );
	sTempMsg	:= CONCAT( sTempMsg, LREAL_TO_STRING( _F_TcMC_Round( Axis.NcToPlc.SetAcc, 4) ) );
	sTempMsg	:= CONCAT( sTempMsg, ', PosTarget: ' );
	sTempMsg	:= CONCAT( sTempMsg, LREAL_TO_STRING( _F_TcMC_Round( sStartRequest.fPosTarget, 4) ) );
	sTempMsg	:= CONCAT( sTempMsg, ',  VeloRequ: ' );
	sTempMsg	:= CONCAT( sTempMsg, LREAL_TO_STRING( _F_TcMC_Round(sStartRequest.fVeloRequ, 4) ) );
	sTempMsg	:= CONCAT( sTempMsg, ',  Acc: ' );
	sTempMsg	:= CONCAT( sTempMsg, LREAL_TO_STRING( _F_TcMC_Round( sStartRequest.fAcc, 4) ) );
	sTempMsg	:= CONCAT( sTempMsg, ',  Dec: ' );
	sTempMsg	:= CONCAT( sTempMsg, LREAL_TO_STRING( _F_TcMC_Round( sStartRequest.fDec, 4) ) );
	sTempMsg	:= CONCAT( sTempMsg, ',  Jerk: ' );
	sTempMsg	:= CONCAT( sTempMsg, LREAL_TO_STRING( _F_TcMC_Round( sStartRequest.fJerk, 4) ) );
	sTempMsg	:= CONCAT( sTempMsg, ', BufMode: ' );
	sTempMsg	:= CONCAT( sTempMsg, UDINT_TO_STRING(sStartRequest.nBufferMode ) );
	sTempMsg	:= CONCAT( sTempMsg, ',  BlendPos: ' );
	sTempMsg	:= CONCAT( sTempMsg, LREAL_TO_STRING( _F_TcMC_Round( sStartRequest.fBlendingPosition, 4) ) );
	sTempMsg	:= CONCAT( sTempMsg, ',  ADS-Stamp: ' );
	sTempMsg	:= CONCAT( sTempMsg, UDINT_TO_STRING( fbAdsReadWrite.fbAdsRdWrt.STAMP_I) );
	IF Axis.PlcToNc.Reserved1 <> 0 THEN (* additional PLC debug info for Beckhoff debugging programs *)
		sTempMsg 	:= CONCAT( sTempMsg, ', PLC-Code=' );
		sTempMsg 	:= CONCAT( sTempMsg, DWORD_TO_STRING(PlcDebugCode) );
	END_IF
	IF Error THEN
		ADSLOGSTR( ADSLOG_MSGTYPE_ERROR + ADSLOG_MSGTYPE_LOG, sTempMsg, '' );		(* vom Typ <Fehlermeldung> *)
	ELSIF CommandAborted THEN
		ADSLOGSTR( ADSLOG_MSGTYPE_WARN, sTempMsg, '' ); 		(* vom Typ <Warnungsmeldung> *)
	ELSE
		ADSLOGSTR( ADSLOG_MSGTYPE_HINT, sTempMsg, '' ); 			(* vom Typ <Hinweismeldung> *)
	END_IF
END_IF
END_ACTION
ACTION ActMonitorContinousMotion:
(*
 * 	monitor continous motion
 *
 * 	monitor UNTIL the axis is in velocity AND the Execute-Input is FALSE
 * 	used with MoveVelocity and other continous commands
*)
IF F_AxisInErrorState(StateDWord := Axis.NcToPlc.StateDWord) THEN (* error while positioning *)
	Error := TRUE;
	ErrorID := Axis.NcToPlc.ErrorCode;
	iState := STATE_INITIALIZATION;
ELSIF NOT F_AxisHasJob(Axis.NcToPlc.StateDWord) OR F_AxisHasBeenStopped(Axis.NcToPlc.StateDWord) THEN (* KSt 27.5.03 *)
	(* aborted during accelertion *)
	CommandAborted := TRUE;
	iState := STATE_INITIALIZATION;
ELSIF InVelocity AND NOT Execute THEN
	(* end of axis control after beeing in velocity for at least one cycle *)
	iState := STATE_INITIALIZATION;
ELSIF Axis.NcToPlc.AxisState = TCNC_PHASE_VELOCONST THEN
	InVelocity := TRUE;
ELSIF InVelocity AND NOT F_AxisIsCompensating(Axis.NcToPlc.StateDWord) THEN
	(* axis was InVelocity but isn't any more, superposition is allowed but *)
	(* any other reason is an abortion *)
	CommandAborted := TRUE;
	iState := STATE_INITIALIZATION;
END_IF
Done := InVelocity;
END_ACTION
ACTION ActMonitorDiscreteMotion:
(*
 * 	monitor discrete motion 
 *
 *	monitor until the target position is reached 
 * 	used with MC_MoveAbsolute and other discrete commands
*)

(* check for reached target position *)
IF (Axis.NcToPlc.OpModeDWord AND  OpMode.TargetPosControl) > 0 THEN (* Target position controlling and PEH enabled ? *)
	IF NOT F_AxisHasJob(Axis.NcToPlc.StateDWord) AND F_AxisIsAtTargetPosition(Axis.NcToPlc.StateDWord) THEN
		Done := TRUE;
		iState := STATE_INITIALIZATION;
	END_IF
ELSE
	IF (Axis.NcToPlc.OpModeDWord AND OpMode.PosAreaControl) > 0 THEN (* Target position controlling enabled ? *)
		IF NOT F_AxisHasJob(Axis.NcToPlc.StateDWord) AND F_AxisInPositionWindow(Axis.NcToPlc.StateDWord) THEN
			Done := TRUE;
			iState := STATE_INITIALIZATION;
		END_IF
	ELSE
		IF NOT F_AxisHasJob(Axis.NcToPlc.StateDWord) THEN
			Done := TRUE;
			iState := STATE_INITIALIZATION;
		END_IF
	END_IF
END_IF;
(* check for timeout *)
IF NOT done AND NOT F_AxisHasJob(Axis.NcToPlc.StateDWord) THEN
	fbTimeOut(IN:= TRUE, PT:= TcMcGlobal.tTargetPosTimeOut);
	IF fbTimeOut.Q THEN
		Error := TRUE;
		ErrorID := MC_ERROR_TARGETPOS_TIMEOUT;
		iState := STATE_INITIALIZATION;
	END_IF;
END_IF;

(* error while positioning *)
IF	F_AxisInErrorState(Axis.NcToPlc.StateDWord) THEN
	Error := TRUE;
	ErrorID := Axis.NcToPlc.ErrorCode;
	iState := STATE_INITIALIZATION;
ELSIF 	F_AxisHasBeenStopped(Axis.NcToPlc.StateDWord)
		AND NOT F_AxisHasJob(Axis.NcToPlc.StateDWord)
		AND NOT (StartType=TCNC_START_HALT)
		AND NOT (StartType=TCNC_START_STOPANDLOCK)
		THEN
		(* manual stop or stop FB ? *)
		ErrorID := MC_ERROR_AXIS_HAS_BEEN_STOPPED;
		CommandAborted 	:= TRUE;
		iState := STATE_INITIALIZATION;
(*	bit 18 is not implemented - 20080610 KSt
ELSIF  F_AxisIsNotInTargetPosition(Axis.NcToPlc.StateDWord) THEN
	( target pos can NOT be reached )
		ErrorID := MC_ERROR_TARGETPOS_TIMEOUT;
		Error := TRUE;
		iState := STATE_INITIALIZATION;
*)
END_IF
END_ACTION
ACTION ActMonitorStop:
(*
 * 	monitor a motion stop or halt
 *
 *	monitor until the target position is reached 
 * 	used with MC_MoveAbsolute and other discrete commands
*)

(* check for deceleration *)
fbTimeOut(IN:= Axis.NcToPlc.AxisState <> TCNC_PHASE_ACCNEG , PT:= TcMcGlobal.tTargetPosTimeOut);

(* error while positioning *)
IF	F_AxisInErrorState(Axis.NcToPlc.StateDWord) THEN
	Error := TRUE;
	ErrorID := Axis.NcToPlc.ErrorCode;
	iState := STATE_INITIALIZATION;

(* check for end of motion  *)
ELSIF NOT F_AxisHasJob(Axis.NcToPlc.StateDWord) THEN
	Done := TRUE;
	iState := STATE_INITIALIZATION;

(* check for timeout *)
ELSIF fbTimeOut.Q THEN
	Error := TRUE;
	ErrorID := MC_ERROR_TARGETPOS_TIMEOUT;
	iState := STATE_INITIALIZATION;
END_IF;
END_ACTION
ACTION ActNcCycleCounter:
(*
	check if cyclic NcToPlc interface changed.
	If not, any Error or CommandAborted condition will be delayed.
	This piece of code prevents from errors if the Plc is called faster than the NC.
	2009-12-08 KSt
*)

fbTimeOut( IN := NcMappingCounter=0, PT:= t#50ms );	(* timout if no nc cyclic feedback for a while *)

NcCycleCounter := DWORD_TO_BYTE(SHR(Axis.NcToPlc.OpModeDWord, 24));
IF NcCycleCounter <> LastNcCycleCounter THEN
	NcMappingCounter := NcMappingCounter + 1; (* has been reset when the command was initiated *)
	NcCycleCounterAvailable := TRUE; (* marked as available when first time not zero - this flag will never be reset at run-time *)
	NcCycleCounterNotAvailable := FALSE;
ELSIF NOT NcCycleCounterAvailable AND fbTimeOut.Q THEN
	NcCycleCounterNotAvailable := TRUE; (* not available on old target systems *)
END_IF
LastNcCycleCounter:=NcCycleCounter;

IF NcCycleCounterNotAvailable OR (NcMappingCounter > 1) OR fbTimeOut.Q THEN
	(*	NcMappingCounter is set to TRUE after an ADS command has been answered.
		NcCyclicFeedbackExpected is set to TRUE when the NcMappingCounter has been 
		incremented at least twice after an ADS command.
		Also TRUE when cycle counter is not available on old target systems and after a time-out 
	*)
	(* 	If NcCyclicFeedbackExpected is false any wrong condition detected from the
		cyclic NcToPlc interface cannot lead to an Error or CommandAborted result.
	*)
	NcCyclicFeedbackExpected := TRUE;
END_IF
END_ACTION

(* POU F_AxisInProtectedMode, ST *)
FUNCTION F_AxisInProtectedMode  : BOOL
(* 	reference: 	NC -> PLC axis interface (128 bytes)
	check if bit 5 of an axis StateDWord is set:
	Axis is in a protected operating mode (e.g. as a slave axis, or under axis interpolation)
	Achse ist in geschützter Betriebsart (z.B. Slave-Achse oder Achsinterpolation)
*)
VAR_INPUT
	StateDWord : DWORD;
END_VAR
VAR
END_VAR
F_AxisInProtectedMode := (StateDWord AND 2#0000_0000_0000_0000_0000_0000_0010_0000) <> 0;
END_FUNCTION

(* POU F_AxisIsReady, ST *)
FUNCTION F_AxisIsReady : BOOL
(* 	reference: 	NC -> PLC axis interface (128 bytes)
	check if bit 0 of an axis StateDWord is set:
	Axis is ready for operation
	Achse ist betriebsbereit
*)
VAR_INPUT
	StateDWord : DWORD;
END_VAR
VAR
END_VAR
F_AxisIsReady := (StateDWord AND 2#0000_0000_0000_0000_0000_0000_0000_0001) <> 0;
END_FUNCTION

(* POU F_AxisIsCompensating, ST *)
FUNCTION F_AxisIsCompensating  : BOOL
(* 	reference: 	NC -> PLC axis interface (128 bytes)
	check if bit 13 of an axis StateDWord is set:
 	After a "Distance Compensation" is startet this beat means:
	Axis is in compensation mode
*)
VAR_INPUT
	StateDWord : DWORD;
END_VAR
VAR
END_VAR
F_AxisIsCompensating := (StateDWord AND 2#0000_0000_0000_0000_0010_0000_0000_0000) <> 0;
END_FUNCTION

(* POU MC_MoveAbsolute, FBD *)
FUNCTION_BLOCK MC_MoveAbsolute
(*	This Function Block commands a controlled motion to a specified absolute position.	*)
VAR_IN_OUT
	Axis				:	AXIS_REF;	(* B *)
END_VAR
VAR_INPUT
	Execute			:	BOOL;	(* B *)	(* Start the motion at rising edge *)
	Position			:	LREAL;	(* B *)	(* Target position for the motion *)
	Velocity			:	LREAL;	(* E *)	(* Value of the maximum velocity *)
	Acceleration		:	LREAL;	(* E *)	(* Value of the maximum acceleration *)
	Deceleration		:	LREAL;	(* E *)	(* Value of the maximum deceleration *)
	Jerk				:	LREAL;	(* E *)	(* Value of the maximum jerk *)
(*	Direction			:	MC_Direction;*)	(* E *)	(* not available *)
	BufferMode		:	MC_BufferMode;	(* E *)
	Options			: 	ST_MoveOptions;	(* V *)	(* optional parameters *)
END_VAR
VAR_OUTPUT
	Done			:	BOOL;	(* B *)
	Busy			: 	BOOL;	(* E *)
	Active			: 	BOOL;	(* E *)
	CommandAborted	:	BOOL;	(* E *)
	Error			:	BOOL;	(* B *)
	ErrorID			:	UDINT;	(* E *)
END_VAR
VAR
	LastExecutionResult: 	_ST_FunctionBlockResults;
	ADSbusy		: 	BOOL;
	MoveGeneric		: 	_FB_MoveUniversalGeneric;
	CmdNo: UINT;
END_VAR
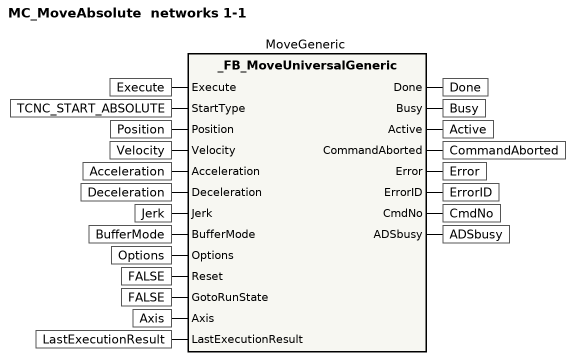
_FBD_ (* Function Block Diagram *)
NETWORK 1
	MoveGeneric :_FB_MoveUniversalGeneric(Execute: Execute, StartType: TCNC_START_ABSOLUTE, Position: Position, Velocity: Velocity, Acceleration: Acceleration, Deceleration: Deceleration, Jerk: Jerk, BufferMode: BufferMode, Options: Options, Reset: FALSE, GotoRunState: FALSE, Axis: Axis, LastExecutionResult: LastExecutionResult, Busy => Busy, Active => Active, CommandAborted => CommandAborted, Error => Error, ErrorID => ErrorID, CmdNo => CmdNo, ADSbusy => ADSbusy) => Done
_END_FBD_
(* the same logic as Structured Text *)
(* Network 1 *)
MoveGeneric (Execute := Execute, StartType := TCNC_START_ABSOLUTE, Position := Position, Velocity := Velocity, Acceleration := Acceleration, Deceleration := Deceleration, Jerk := Jerk, BufferMode := BufferMode, Options := Options, Reset := FALSE, GotoRunState := FALSE, Axis := Axis, LastExecutionResult := LastExecutionResult);
Busy := MoveGeneric .Busy;
Active := MoveGeneric .Active;
CommandAborted := MoveGeneric .CommandAborted;
Error := MoveGeneric .Error;
ErrorID := MoveGeneric .ErrorID;
CmdNo := MoveGeneric .CmdNo;
ADSbusy := MoveGeneric .ADSbusy;
Done := MoveGeneric .Done;
END_FUNCTION_BLOCK

(* POU F_AxisIsAtTargetPosition, ST *)
FUNCTION F_AxisIsAtTargetPosition  : BOOL
(* 	reference: 	NC -> PLC axis interface (128 bytes)
	check if bit 4 of an axis StateDWord is set:
	Axis is at target position (PEH) (physical feedback)
	Achse ist in Zielposition (PEH) (physik. Rückmeldung)
*)
VAR_INPUT
	StateDWord : DWORD;
END_VAR
VAR
END_VAR
F_AxisIsAtTargetPosition := (StateDWord AND 2#0000_0000_0000_0000_0000_0000_0001_0000) <> 0;
END_FUNCTION

(* POU F_AxisInPositionWindow, ST *)
FUNCTION F_AxisInPositionWindow : BOOL
(* 	reference: 	NC -> PLC axis interface (128 bytes)
	check if bit 3 of an axis StateDWord is set:
	Axis is in position window (physical feedback)
	Achse ist im Positionsbereichsfenster (physik. Rückmeldung) 
*)
VAR_INPUT
	StateDWord : DWORD;
END_VAR
VAR
END_VAR
F_AxisInPositionWindow := (StateDWord AND 2#0000_0000_0000_0000_0000_0000_0000_1000) <> 0;
END_FUNCTION

(* POU _FB_ReadWriteParameter, ST *)
{library private}
FUNCTION_BLOCK _FB_ReadWriteParameter
VAR_IN_OUT
	Axis				:	AXIS_REF;
END_VAR
VAR_INPUT
	Enable			:	BOOL;
	ParameterNumber	:	MC_AxisParameter;
	Mode			:	INT; 		(* read/write *)
	ParameterType	:	INT;		(* bool/ not  bool *)
END_VAR
VAR_OUTPUT
	Done			:	BOOL;
	Busy: BOOL;
	Error			:	BOOL;
	ErrorID			:	UDINT;
	ADSbusy: BOOL;
END_VAR
VAR_IN_OUT
	ValueLreal		:	LREAL;
	ValueDword		:	DWORD;
	ValueBool		:	BOOL;
END_VAR
VAR
	iState			:	_E_TcMC_STATES := STATE_INITIALIZATION;
	fbAdsRead		:	ADSREAD;
	fbAdsWrite		:	ADSWRITE;

	dwValue			:	DWORD;
	lrValue			:	ARRAY[1..10] OF LREAL;
	NcBoolValue		:	UINT;

	bStarted			:	BOOL;
	stParaStruct		:	_ST_ParaStruct;
	n: INT;
	i: INT;
END_VAR
VAR CONSTANT
(*	ParaDWORD		:	INT:= 1;*)
	ParaLREAL		:	INT := 2;
(*	ParaBOOL		:	INT := 3;*)
END_VAR
(* ====================================================================== *)
(* *)
(* ====================================================================== *)

CASE iState OF
STATE_INITIALIZATION:	(* Ruhezustand *)
	Busy := FALSE;
    	IF Enable THEN
		(* initialize output values *)
		Done := FALSE;
		Error := FALSE;
		ErrorID := 0;

		stParaStruct.LrealSize := SIZEOF(lrValue[1]);
		stParaStruct.LrealOffset := 1;

		(* some parameters are read immediately out of the cyclic axis interfaces *)
		(* other parameters are read via ADS, F_GetIndexGroup finds the required ADS parameters in this case *)
		IF Mode=READWRITEPARAMETERMODE_READ THEN
			CASE ParameterNumber OF
				CommandedPosition :
					stParaStruct.IndexOffset := 16#0000_0000;
					stParaStruct.IndexGroup := 0;
					stParaStruct.ParaType := ParaLreal;
					ValueLreal := Axis.NcToPlc.SetPos;
					Done := TRUE;
				ActualVelocity:
					stParaStruct.IndexOffset := 16#0000_0000;
					stParaStruct.IndexGroup := 0;
					stParaStruct.ParaType := ParaLreal;
					ValueLreal := Axis.NcToPlc.ActVelo;
					Done := TRUE;
				CommandedVelocity:
					stParaStruct.IndexOffset := 16#0000_0000;
					stParaStruct.IndexGroup := 0;
					stParaStruct.ParaType := ParaLreal;
					ValueLreal := Axis.NcToPlc.SetVelo;
					Done := TRUE;
				ELSE
					(* check index offset *)
					stParaStruct := _F_GetIndexGroup(ParaNumber := ParameterNumber, Mode:=Mode);
			END_CASE;
		ELSE
			(* check index offset *)
			stParaStruct := _F_GetIndexGroup(ParaNumber := ParameterNumber, Mode:=Mode);
		END_IF
		IF NOT Done THEN
			Busy := TRUE;
			iState := STATE_ORDER;
		END_IF
	ELSE
		Done := FALSE; (* reset with Enable=FALSE *)
		Error := FALSE;			(* reset at falling edge of Execute *)
		ErrorID := 0;
	END_IF
END_CASE

CASE iState OF
STATE_INITIALIZATION:
	;	(* already done before *)
STATE_ORDER :
		(* read via ADS *)
		IF FALSE AND (stParaStruct.ParaType <> ParameterType) (* no check !!*)
		THEN
			(* type mismatch *)
			Done := FALSE;
			ErrorID := MC_ERROR_COMMAND_NOT_ALLOWED;
			Error := TRUE;
		ELSIF stParaStruct.ParaType <> PARAMETERTYPE_NOTYPE THEN
			CASE Mode OF
(*------------------ Read parameter ---------------------------------------------------------------*)
				READWRITEPARAMETERMODE_READ	:
					CASE stParaStruct.ParaType OF
						PARAMETERTYPE_DWORD :	(* read DWORD *)
							fbAdsRead(	NETID:= TcMcGlobal.NCNETID_TCMC,
								PORT:= TcMcGlobal.NCPORT_TCMC,
								IDXGRP:= stParaStruct.IndexGroup+Axis.NcToPlc.AxisId,
								IDXOFFS:= stParaStruct.IndexOffset,
								LEN:= SIZEOF(dwValue),
								DESTADDR:= ADR(dwValue),
								READ:= TRUE,
								TMOUT:= TcMcGlobal.tADSTimeOut);
								ValueDword := DWORD_TO_DINT(dwValue);
								ValueLreal := DWORD_TO_REAL (dwValue);
								ValueBool := DWORD_TO_BOOL(dwValue);

						PARAMETERTYPE_LREAL :		(* read LREAL *)
							fbAdsRead(	NETID:= TcMcGlobal.NCNETID_TCMC,
								PORT:= TcMcGlobal.NCPORT_TCMC,
								IDXGRP:= stParaStruct.IndexGroup+Axis.NcToPlc.AxisId,
								IDXOFFS:= stParaStruct.IndexOffset,
								LEN:= MIN(SIZEOF(lrValue), stParaStruct.LrealSize),
								DESTADDR:= ADR(lrValue),
								READ:= TRUE,
								TMOUT:=  TcMcGlobal.tADSTimeOut);
								ValueLreal := lrValue[stParaStruct.LrealOffset];
								IF ValueLreal > 16#FFFF_FFFF THEN	(* 31.5.2007 KSt - avoid FPU exception *)
									ValueDword := 0;
									ValueBool := TRUE;
								ELSIF ValueLreal < -16#8000_0000 THEN 	(* 31.5.2007 KSt - avoid FPU exception *)
									ValueDword := 0;
									ValueBool := TRUE;
								ELSE
									ValueDword := LREAL_TO_DINT(lrValue[stParaStruct.LrealOffset]); 	(* 31.5.2007 KSt - existing code *)
									ValueBool := LREAL_TO_BOOL(lrValue[stParaStruct.LrealOffset]);		(* 31.5.2007 KSt - existing code *)
								END_IF

						PARAMETERTYPE_BOOL :		(* read bool *)
							fbAdsRead(	NETID:= TcMcGlobal.NCNETID_TCMC,
								PORT:= TcMcGlobal.NCPORT_TCMC,
								IDXGRP:= stParaStruct.IndexGroup+Axis.NcToPlc.AxisId,
								IDXOFFS:= stParaStruct.IndexOffset,
								LEN:= SIZEOF(NcBoolValue),
								DESTADDR:= ADR(NcBoolValue),
								READ:= TRUE,
								TMOUT:=  TcMcGlobal.tADSTimeOut);
								ValueBool := UINT_TO_BOOL(NcBoolValue);
								ValueDword := UINT_TO_DINT(NcBoolValue);
								ValueLreal := UINT_TO_LREAL (NcBoolValue);

					END_CASE;
(*------------------ Write parameter ---------------------------------------------------------------*)
				READWRITEPARAMETERMODE_WRITE	:
					CASE stParaStruct.ParaType OF
						PARAMETERTYPE_DWORD:	(* read DWORD *)
							ValueDword := LREAL_TO_DWORD(ValueLreal);
							fbAdsWrite(	NETID:= TcMcGlobal.NCNETID_TCMC,
								PORT:= TcMcGlobal.NCPORT_TCMC,
								IDXGRP:= stParaStruct.IndexGroup+Axis.NcToPlc.AxisId,
								IDXOFFS:= stParaStruct.IndexOffset,
								LEN:= SIZEOF(ValueDword),
								SRCADDR:= ADR(ValueDword),
								WRITE:= TRUE,
								TMOUT:= TcMcGlobal.tADSTimeOut);

						PARAMETERTYPE_LREAL :		(* read LREAL *)
							n := SIZEOF(lrValue) / SIZEOF(lrValue[1]);
							FOR i := 1 TO n DO lrValue[i] := 0; END_FOR
							lrValue[stParaStruct.LrealOffset] := ValueLreal;
							fbAdsWrite(	NETID:= TcMcGlobal.NCNETID_TCMC,
								PORT:= TcMcGlobal.NCPORT_TCMC,
								IDXGRP:= stParaStruct.IndexGroup+Axis.NcToPlc.AxisId,
								IDXOFFS:= stParaStruct.IndexOffset,
								LEN:= MIN(SIZEOF(lrValue), stParaStruct.LrealSize),
								SRCADDR:= ADR(lrValue),
								WRITE:= TRUE,
								TMOUT:=  TcMcGlobal.tADSTimeOut);

						PARAMETERTYPE_BOOL :		(* read BOOL *)
							NcBoolValue := BOOL_TO_UINT(ValueBool);
							fbAdsWrite(	NETID:= TcMcGlobal.NCNETID_TCMC,
								PORT:= TcMcGlobal.NCPORT_TCMC,
								IDXGRP:= stParaStruct.IndexGroup+Axis.NcToPlc.AxisId,
								IDXOFFS:= stParaStruct.IndexOffset,
								LEN:= SIZEOF(NcBoolValue),
								SRCADDR:= ADR(NcBoolValue),
								WRITE:= TRUE,
								TMOUT:=  TcMcGlobal.tADSTimeOut);
					END_CASE;
			END_CASE;

